// TwinCAT 3 PLC project RBB
// ProgramVersion: 3.1.4024.0
// libraries:
//   Tc2_Standard, * (Beckhoff Automation GmbH)
//   Tc2_System, * (Beckhoff Automation GmbH)
//   Tc3_Module, * (Beckhoff Automation GmbH)
// project tree:
//   DUTs/ E_ClientServerSteps.TcDUT, GPSReceive.TcDUT, ST_FrameFifoEntry.TcDUT, ST_FrameFifoEntrydata.TcDUT, ST_FrameFifoEntrydatarx.TcDUT, ST_FrameFifoEntrydata_1.TcDUT, ST_FrameFifoEntrydata_2.TcDUT, Union_LREAL.TcDUT, Union_LREAL_STRING.TcDUT, Union_REAL.TcDUT, Union_STRING_10.TcDUT, Union_STRING_2.TcDUT, Union_STRING_3.TcDUT, Union_STRING_4.TcDUT, Union_UDINT.TcDUT, Union_UINT.TcDUT, Union_WORD.TcDUT
//   GVLs/ GVL.TcGVL
//   / PlcTask.TcTTO
//   POUs/Background/ Background.TcPOU
//   POUs/Communication/ FB_AHRSCommunication.TcPOU, FB_ESCcommunication.TcPOU, FB_GPSCommunication.TcPOU
//   POUs/FUCTION BLOCK/UDP Source/ FB_FrameFifo.TcPOU, FB_FrameFiforx.TcPOU, FB_FrameFifo_1.TcPOU, FB_FrameFifo_2.TcPOU, FB_LogFifo.TcPOU, FB_PeerToPeer.TcPOU, FB_PeerToPeer_1.TcPOU, FB_PeerToPeer_2.TcPOU
//   POUs/FUNCTION/ FC_AnalogRead.TcPOU, FC_BatCalculate.TcPOU, FC_CalculateAzimuth.TcPOU, FC_HaversineDistance.TcPOU, FC_HMIRead.TcPOU
//   POUs/ MAIN.TcPOU, UDPCommunication_RBB.TcPOU
//   POUs/Module/ ESC.TcPOU, RelayModule.TcPOU
//   POUs/Sensor/ AHRS.TcPOU, GPS.TcPOU, LeakSensor.TcPOU
// real-time tasks:
//   TASK PlcTask: cycle T#10ms, priority 20, ADS port 350

CONFIGURATION RBB
    RESOURCE PLC ON TwinCAT3
        TASK PlcTask(INTERVAL := T#10ms, PRIORITY := 20);
        PROGRAM MAIN WITH PlcTask : MAIN;
    END_RESOURCE
END_CONFIGURATION

// ---- DUTs/E_ClientServerSteps.TcDUT
TYPE E_ClientServerSteps :
(
	eUDP_STATE_IDLE		:= 0,
	eUDP_STATE_CREATE_START,
	eUDP_STATE_CREATE_WAIT,
	eUDP_STATE_SEND_START,
	eUDP_STATE_SEND_WAIT,
	eUDP_STATE_RECEIVE_START,
	eUDP_STATE_RECEIVE_WAIT,
	eUDP_STATE_CLOSE_START,
	eUDP_STATE_CLOSE_WAIT,
	eUDP_STATE_ERROR
);
END_TYPE

// ---- DUTs/GPSReceive.TcDUT
TYPE GPSReceive :
UNION
	value : STRING;
	packed : ARRAY[0..69] OF BYTE;
END_UNION
END_TYPE

// ---- DUTs/ST_FrameFifoEntry.TcDUT
TYPE ST_FrameFifoEntry :
STRUCT
	 caseSelector : INT;              // Selector to choose the active structure
    data         : U_FrameFifoEntrydata;
END_STRUCT
END_TYPE

// ---- DUTs/ST_FrameFifoEntrydata.TcDUT
TYPE ST_FrameFifoEntrydata :
STRUCT
	stRemoteAddr 	: ST_SockAddr;
	txdata : ARRAY[0..TXDATASIZE] OF BYTE;	
END_STRUCT
END_TYPE

// ---- DUTs/ST_FrameFifoEntrydatarx.TcDUT
TYPE ST_FrameFifoEntrydatarx :
STRUCT
	stRemoteAddr 	: ST_SockAddr;
	rxdata : ARRAY[0..RXDATASIZE] OF BYTE;
END_STRUCT
END_TYPE

// ---- DUTs/ST_FrameFifoEntrydata_1.TcDUT
TYPE ST_FrameFifoEntrydata_1 :
STRUCT	
	stRemoteAddr 	: ST_SockAddr;
	txdata : ARRAY[0..TXDATASIZE_1] OF BYTE; 
END_STRUCT
END_TYPE

// ---- DUTs/ST_FrameFifoEntrydata_2.TcDUT
TYPE ST_FrameFifoEntrydata_2 :
STRUCT
	stRemoteAddr 	: ST_SockAddr;
	txdata : ARRAY[0..TXDATASIZE_2] OF BYTE; 
END_STRUCT
END_TYPE

// ---- DUTs/Union_LREAL.TcDUT
TYPE Union_LREAL :
UNION
	value : LREAL;
	packed : ARRAY[0..7] OF BYTE;
END_UNION
END_TYPE

// ---- DUTs/Union_LREAL_STRING.TcDUT
TYPE Union_LREAL_STRING :
UNION
	value : STRING;
	packed : ARRAY[0..7] OF BYTE;
END_UNION
END_TYPE

// ---- DUTs/Union_REAL.TcDUT
TYPE Union_REAL :
UNION
	value : REAL;
	Packed : ARRAY[0..3] OF BYTE;
END_UNION
END_TYPE

// ---- DUTs/Union_STRING_10.TcDUT
TYPE Union_STRING_10 :
UNION
	value : STRING;
	Packed : ARRAY[0..9] OF BYTE;
END_UNION
END_TYPE

// ---- DUTs/Union_STRING_2.TcDUT
TYPE Union_STRING_2 :
UNION
	value : STRING;
	Packed : ARRAY[0..1] OF BYTE;
END_UNION
END_TYPE

// ---- DUTs/Union_STRING_3.TcDUT
TYPE Union_STRING_3 :
UNION
	value : STRING;
	Packed : ARRAY[0..2] OF BYTE;
END_UNION
END_TYPE

// ---- DUTs/Union_STRING_4.TcDUT
TYPE Union_STRING_4 :
UNION
	value : STRING;
	Packed : ARRAY[0..3] OF BYTE;
END_UNION
END_TYPE

// ---- DUTs/Union_UDINT.TcDUT
TYPE Union_UDINT :
UNION
	value : UDINT ;
	packed : ARRAY[0..3] OF BYTE;
END_UNION
END_TYPE

// ---- DUTs/Union_UINT.TcDUT
TYPE Union_UINT :
UNION
	value : UINT;
	packed : ARRAY[0..1] OF BYTE;
END_UNION
END_TYPE

// ---- DUTs/Union_WORD.TcDUT
TYPE Union_WORD :
UNION
	value : WORD;
	packed : ARRAY[0..1] OF BYTE;
END_UNION
END_TYPE

// ---- GVLs/GVL.TcGVL
VAR_GLOBAL
	
	RxBufferEL6001		: ComBuffer;	
	TxBufferEL6001		: ComBuffer;	
	
	RxBufferEL6002	    : ComBuffer;	
	TxBufferEL6002		: ComBuffer;	
	
	RxBufferEL6021		: ComBuffer;	
	TxBufferEL6021		: ComBuffer;
	
	
	AI_00 AT%I* : WORD;
    AI_01 AT%I* : WORD;
	
	//Algorithm_Sw : BOOL;
 
 
	 
END_VAR

VAR_GLOBAL CONSTANT
 TXDATASIZE : INT := 101; // 59(60) , 23(24) , 17(18) , 101(102) , test 105(106)
 
 TXDATASIZE_1 : INT := 12; 
 TXDATASIZE_2 : INT := 15; 
 
 
 RXDATASIZE : INT := 1000; 
 
 
 PLCPRJ_BUFFER_SIZE					: UDINT := 1000;(* Max. internal fifo/receiver buffer size *)

(* Some project specific error codes *)
PLCPRJ_ERROR_SENDFIFO_OVERFLOW		: UDINT := 16#8103;
PLCPRJ_ERROR_RECFIFO_OVERFLOW		: UDINT := 16#8104;

END_VAR

// ---- POUs/MAIN.TcPOU
PROGRAM MAIN
VAR

// BAT

rBatvoltage : REAL; // UDP DATA
rBatcurrent : REAL; // UDP DATA
rBatWattsec : LREAL; 
AccumulatedBatData : LREAL :=0.0; // UDP DATA
lbatstate : LREAL; // UDP DATA

battimer : TON;

HMIbatV : STRING; // HMI
HMIbatA : STRING; // HMI
HMIbatW : STRING; // HMI
HMIbatS : STRING; // HMI

//AHRS

bAHRSError : BOOL;
AHRSErrorID : ComError_t;

HMIYAW : STRING;
HMIPITCH : STRING;
HMIROLL : STRING;

// ESC

bESCerror : BOOL;
ESCerrorID : ComError_t;
thrusterrightrpm : UINT;
thrusterleftrpm : UINT;


// GPS

bGPSrror : BOOL;
GPSErrorID : ComError_t;

GPSlat1 : LREAL;
GPSlon1 : LREAL;

HMILatitude : STRING;
HMILongitude : STRING;
HMISpeed : STRING;
	
// LEAK SENSOR

SystemLeakState : BOOL;
Leaksensorerror : BOOL;
Leaksensorerrorid : MODBUS_ERRORS;

// RELAY	
  
RelayModuledata : BYTE ;
RelayModuleError : BOOL;
RelayModuleErrorID : UDINT;

// UDP

UDPAlgorithm : INT;
UDPtimer : TON;


// Algorithm

    state : UINT := 0;
    timer : TON;
    stayTimer : TON;
    distance : LREAL;
    azimuth : LREAL;
   
    lat1, lon1, lat2, lon2, lat3, lon3, lat4, lon4 : LREAL;
	lat5, lon5, lat6, lon6, lat7, lon7, lat8, lon8,
	lat9, lon9, lat10, lon10, lat11, lon11, lat12, lon12,
	lat13, lon13, lat14, lon14, lat15, lon15, lat16, lon16 : LREAL;
	
    baseLat, baseLon : LREAL;
    currentTargetLat, currentTargetLon : LREAL;
    waypointIndex : UINT :=1;
	turnAngle : LREAL;
	turnangelzero : BOOL;
	esccontroltimer : TON;
	esccontroltimer1 : TON;
	esccontroltimer2 : TON;
	esccontroltimer3 : TON;
	esccontroltimer4 : TON;
		
	bturnangle : BOOL := TRUE;
	bturnangle2 : BOOL := TRUE;
	bstraight : BOOL := TRUE;
	bstop : BOOL := TRUE;
	
// Utilities

	bPCShutdown: BOOL;
	fbShutdown: NT_Shutdown;
	bShutdown: BOOL :=FALSE;
	
	step : INT;
	start : BOOL;
	Shutdown : BOOL := FALSE;
	
	i: INT;
END_VAR

// BAT 

rBatvoltage := FC_AnalogRead(selectData := AI_00, SelectRange := 600);
rBatcurrent := FC_AnalogRead(selectData := AI_01, SelectRange := 100);
rBatWattsec := (rBatvoltage*rBatcurrent)/3600;

IF NOT battimer.Q THEN
battimer(IN:=TRUE, PT := T#1S);
ELSE 
battimer(IN:=FALSE);
AccumulatedBatData := AccumulatedBatData + rBatWattsec;
END_IF

lbatstate := FC_BatCalculate(lbatdata := AccumulatedBatData);

HMIbatV := FC_HMIRead(linput := rBatvoltage, inumber := 2);
HMIbatA := FC_HMIRead(linput := rBatcurrent, inumber := 2);
HMIbatW := FC_HMIRead(linput := AccumulatedBatData , inumber := 2);
HMIbatS := FC_HMIRead(linput := lbatstate, inumber := 2);
 
// AHRS 

AHRS();
bAHRSError := AHRS.bAHRSError;
AHRSErrorID := AHRS.AHRSErrorID;

HMIYAW :=FC_HMIRead(linput := AHRS.ResultYAW, inumber := 1);
HMIPITCH :=FC_HMIRead(linput := AHRS.ResultPITCH, inumber := 1);
HMIROLL :=FC_HMIRead(linput := AHRS.ResultROLL, inumber := 1);

// ESC

ESC();
bESCerror := ESC.bESCerror;
ESCerrorID := ESC.ESCerrorID;

IF ESC.sMotorspeed = 'ESC1:1650' THEN
	thrusterrightrpm := 750;
ELSIF ESC.sMotorspeed = 'ESC1:1750' THEN
	thrusterrightrpm := 1250;
ELSIF  ESC.sMotorspeed = 'ESC1:1700' THEN
	thrusterrightrpm := 1000;
ELSIF ESC.sMotorspeed = 'ESC2:1350' THEN
	thrusterleftrpm := 750;
ELSIF  ESC.sMotorspeed = 'ESC2:1250' THEN
	thrusterleftrpm := 1250;
ELSIF  ESC.sMotorspeed = 'ESC2:1300' THEN
	thrusterleftrpm := 1000;
END_IF 


// GPS 

GPS();
bGPSrror := GPS.bGPSrror;
GPSErrorID := GPS.GPSErrorID;

GPSlat1 := GPS.gpslat;
GPSlon1 := GPS.gpslon;

HMILatitude :=FC_HMIRead(linput := GPS.gpslat, inumber := 1);
HMILongitude :=FC_HMIRead(linput := GPS.gpslon, inumber := 1);
HMISpeed :=FC_HMIRead(linput := GPS.gpsSpeedms, inumber := 1);

// LEAK SENSOR

LeakSensor();
SystemLeakState := LeakSensor.LeakSensorState;
Leaksensorerror := LeakSensor.Leaksensorerror;
Leaksensorerrorid := LeakSensor.leaksensorerrorid;
 
// RELAY Module

RelayModule();
RelayModuleError := RelayModule.RelayModuleError;
RelayModuleErrorID := RelayModule.RelayModuleErrorID;
RelayModuledata := RelayModule.relaymodulesendOnData;

// UDPCommunication

UDPCommunication_RBB();
	CASE UDPAlgorithm OF
		0 :
		IF UDPCommunication_RBB.UDPstart THEN
			IF UDPCommunication_RBB.Receiveaddress = 16#01 THEN
				UDPAlgorithm := 10;
			ELSIF UDPCommunication_RBB.Receiveaddress = 16#02 THEN
				UDPAlgorithm := 10;
			ELSIF UDPCommunication_RBB.Receiveaddress = 16#03 THEN
				UDPAlgorithm := 10;
			ELSIF UDPCommunication_RBB.Receiveaddress = 16#04 THEN
				UDPAlgorithm := 10;
			END_IF		
		END_IF
		
		10 :
		 UDPCommunication_RBB.UDPstart := FALSE;
		 UDPtimer(IN:= TRUE, PT:= T#1S);
		 IF UDPtimer.Q THEN
		 UDPCommunication_RBB.UDPstart3 := TRUE;
		 UDPtimer(IN:= FALSE);
		 UDPAlgorithm := 20;
		 END_IF
		 		 		 
		 20 :
		 UDPtimer(IN:= TRUE, PT:= T#1S);
		 IF UDPtimer.Q THEN
		 UDPCommunication_RBB.UDPstart3 := FALSE;	
         UDPtimer(IN:= FALSE);
		 UDPAlgorithm := 30; 
		 END_IF
		 		 
		 30 : 
		 UDPtimer(IN:= TRUE, PT:= T#1S);
		 IF UDPtimer.Q THEN
		  IF UDPCommunication_RBB.Receiveaddress = 16#03 THEN
			UDPCommunication_RBB.UDPstart2 := TRUE;
			UDPtimer(IN:= FALSE);
		    UDPAlgorithm := 40;
		  ELSE
		  UDPCommunication_RBB.UDPstart := TRUE;		
		  UDPCommunication_RBB.bSendOnceToRemote2 := FALSE;
		  UDPtimer(IN:= FALSE);
		  UDPAlgorithm := 0;
		  END_IF
		 END_IF
		 
		 40 :
		 UDPtimer(IN:= TRUE, PT:= T#1S);
		 IF UDPtimer.Q THEN
		 UDPCommunication_RBB.UDPstart2 := FALSE;	
         UDPtimer(IN:= FALSE);
		 UDPAlgorithm := 50; 
		 END_IF
		 
		 50 :
		 UDPtimer(IN:= TRUE, PT:= T#1S);
		 IF UDPtimer.Q THEN
		 UDPCommunication_RBB.UDPstart := TRUE;
		 UDPCommunication_RBB.bSendOnceToRemote1 := FALSE;
		 UDPtimer(IN:= FALSE);
		 UDPAlgorithm := 0;
		 END_IF
	END_CASE


// Algorithm

IF UDPCommunication_RBB.Algorithmstop THEN	

  IF UDPCommunication_RBB.Algorithm_Sw THEN
    CASE state OF
        0: // Start algorithm, initialize first target
		    lat1 := UDPCommunication_RBB.packetwetpointlat1.value;
			lon1 := UDPCommunication_RBB.packetwetpointlot1.value;
            currentTargetLat := lat1;
            currentTargetLon := lon1;
            state := 10;
			

        10: // Calculate distance to the current target
            distance := FC_HaversineDistance(GPS.gpslat, GPS.gpslon, currentTargetLat, currentTargetLon);
            IF ABS(distance) <=10 THEN
                state := 13; // Go to the stay state if already within 10m
            ELSE
                timer(IN := TRUE, PT := T#1S);
                IF timer.Q THEN
                    state := 11;
                    timer(IN := FALSE); // Reset timer
                END_IF
            END_IF

        11: // Calculate azimuth and move
            azimuth := FC_CalculateAzimuth(GPS.gpslat, GPS.gpslon, currentTargetLat, currentTargetLon);
            turnAngle := azimuth - UDPCommunication_RBB.packetahrsheading.value;
			
            IF turnAngle > 180 THEN
                turnAngle := turnAngle - 360;
            ELSIF turnAngle < -180 THEN
                turnAngle := turnAngle + 360;
            END_IF
			
			IF ABS(turnAngle) <= 25 THEN  
                 state := 12; 
											
            ELSIF turnAngle > 0 THEN// Turn right
			   IF bturnangle THEN
				ESC.sMotorspeed := 'ESC2:1250'; //62.5%
				esccontroltimer2(IN:=TRUE, PT:=T#1S);
				 IF esccontroltimer2.Q THEN
				   ESC.sMotorspeed := 'ESC1:1650';	// 37.5%			   
				   esccontroltimer2(IN:=FALSE);
                   bturnangle := FALSE;				   
				 END_IF 			
				END_IF 
											
            ELSE// Turn left	
				 IF bturnangle2 THEN
				  ESC.sMotorspeed := 'ESC1:1750'; //62.5% 
				 esccontroltimer4(IN:=TRUE, PT:=T#1S);
				  IF esccontroltimer4.Q THEN
				   ESC.sMotorspeed := 'ESC2:1350'; //37.5%
				   esccontroltimer4(IN:=FALSE);
                   bturnangle2 := FALSE;				   
				  END_IF 			
				END_IF 
		  END_IF 
             				        
			
									
		12 : // Move
		
		distance := FC_HaversineDistance(GPS.gpslat, GPS.gpslon, currentTargetLat, currentTargetLon);
		azimuth := FC_CalculateAzimuth(GPS.gpslat, GPS.gpslon, currentTargetLat, currentTargetLon);
        turnAngle := azimuth - UDPCommunication_RBB.packetahrsheading.value;
			
            IF turnAngle > 180 THEN
                turnAngle := turnAngle - 360;
            ELSIF turnAngle < -180 THEN
                turnAngle := turnAngle + 360;
            END_IF
			
			
		
            IF ABS(turnAngle) <= 25 THEN  
			IF bstraight THEN
				ESC.sMotorspeed := 'ESC2:1300'; //50%
				esccontroltimer1(IN:=TRUE, PT:=T#1S);
				 IF esccontroltimer1.Q THEN
				   ESC.sMotorspeed := 'ESC1:1700'; // 50%
				   esccontroltimer1(IN:=FALSE);
                   bstraight := FALSE;				   
				 END_IF 	
                  ELSIF ABS(distance) <=10 THEN		         
				   esccontroltimer3(IN:=TRUE, PT:=T#1S);
				   IF esccontroltimer3.Q THEN	   
				   ESC.sMotorspeed := 'stop';			   
				   esccontroltimer3(IN:=FALSE);				
				   state := 13;	
				   END_IF
			  END_IF  
              ELSE
                   state :=11;	
	               bstraight := TRUE;
				   bturnangle := TRUE;	
				   bturnangle2 := TRUE;	
              END_IF	


        13: // Check distance again
            stayTimer(IN := TRUE, PT := T#30S);
            IF stayTimer.Q THEN
				ESC.sMotorspeed := '';
				   bstraight := TRUE;
				   bturnangle := TRUE;	
				   bturnangle2 := TRUE;	
                state := 14; // Next waypoint or finish
                stayTimer(IN := FALSE); // Reset stay timer
            END_IF
           


        14: // Check if there are more waypoints to visit
		    //waypointIndex 
            CASE waypointIndex OF
                1:
				    lat2 := UDPCommunication_RBB.packetwetpointlat2.value;
					lon2 := UDPCommunication_RBB.packetwetpointlot2.value;
                    currentTargetLat := lat2;
                    currentTargetLon := lon2;
                    waypointIndex := 2;
                    state := 10;
                2:
				    lat3 := UDPCommunication_RBB.packetwetpointlat3.value;
					lon3 := UDPCommunication_RBB.packetwetpointlot3.value;
                    currentTargetLat := lat3;
                    currentTargetLon := lon3;
                    waypointIndex := 3;
                    state := 10;
                3:
				    lat4 := UDPCommunication_RBB.packetwetpointlat4.value;
					lon4 := UDPCommunication_RBB.packetwetpointlot4.value;
                    currentTargetLat := lat4;
                    currentTargetLon := lon4;
                    waypointIndex := 4;
                    state := 10;
                4:
				    lat5 := UDPCommunication_RBB.packetwetpointlat4.value;
					lon5 := UDPCommunication_RBB.packetwetpointlot4.value;
                    currentTargetLat := lat5;
                    currentTargetLon := lon5;
                    waypointIndex := 5;
                    state := 10;
				5:
				    lat6 := UDPCommunication_RBB.packetwetpointlat4.value;
					lon6 := UDPCommunication_RBB.packetwetpointlot4.value;
                    currentTargetLat := lat6;
                    currentTargetLon := lon6;
                    waypointIndex := 6;
                    state := 10;
				6:
				    lat7 := UDPCommunication_RBB.packetwetpointlat4.value;
					lon7 := UDPCommunication_RBB.packetwetpointlot4.value;
                    currentTargetLat := lat7;
                    currentTargetLon := lon7;
                    waypointIndex := 7;
                    state := 10;
				7:
				    lat8 := UDPCommunication_RBB.packetwetpointlat4.value;
					lon8 := UDPCommunication_RBB.packetwetpointlot4.value;
                    currentTargetLat := lat8;
                    currentTargetLon := lon8;
                    waypointIndex := 8;
                    state := 10;
				8:
				    lat9 := UDPCommunication_RBB.packetwetpointlat4.value;
					lon9 := UDPCommunication_RBB.packetwetpointlot4.value;
                    currentTargetLat := lat9;
                    currentTargetLon := lon9;
                    waypointIndex := 9;
                    state := 10;
				9:
				    lat10 := UDPCommunication_RBB.packetwetpointlat4.value;
					lon10 := UDPCommunication_RBB.packetwetpointlot4.value;
                    currentTargetLat := lat10;
                    currentTargetLon := lon10;
                    waypointIndex := 10;
                    state := 10;
				10:
				    lat11 := UDPCommunication_RBB.packetwetpointlat4.value;
					lon11 := UDPCommunication_RBB.packetwetpointlot4.value;
                    currentTargetLat := lat11;
                    currentTargetLon := lon11;
                    waypointIndex := 11;
                    state := 10;
				11:
				    lat12 := UDPCommunication_RBB.packetwetpointlat4.value;
					lon12 := UDPCommunication_RBB.packetwetpointlot4.value;
                    currentTargetLat := lat12;
                    currentTargetLon := lon12;
                    waypointIndex := 12;
                    state := 10;
				12:
				    lat13 := UDPCommunication_RBB.packetwetpointlat4.value;
					lon13 := UDPCommunication_RBB.packetwetpointlot4.value;
                    currentTargetLat := lat13;
                    currentTargetLon := lon13;
                    waypointIndex := 13;
                    state := 10;
				13:
				    lat14 := UDPCommunication_RBB.packetwetpointlat4.value;
					lon14 := UDPCommunication_RBB.packetwetpointlot4.value;
                    currentTargetLat := lat14;
                    currentTargetLon := lon14;
                    waypointIndex := 14;
                    state := 10;
				14:
				    lat15 := UDPCommunication_RBB.packetwetpointlat4.value;
					lon15 := UDPCommunication_RBB.packetwetpointlot4.value;
                    currentTargetLat := lat15;
                    currentTargetLon := lon15;
                    waypointIndex := 15;
                    state := 10;
				15:
				    lat16 := UDPCommunication_RBB.packetwetpointlat4.value;
					lon16 := UDPCommunication_RBB.packetwetpointlot4.value;
                    currentTargetLat := lat16;
                    currentTargetLon := lon16;
                    waypointIndex := 16;
                    state := 10;  
 
                 16 :  
                    state := 20;
            END_CASE	 
                 20: 
		        ESC.sMotorspeed := 'stop';
				 
	 			
    END_CASE
ELSE
    // Reset state and timers if Algorithm_sw is turned off
    state := 0;
    timer(IN := FALSE);
    stayTimer(IN := FALSE);
    waypointIndex := 1; // Reset waypoint index
END_IF 

ELSE
	esc.sMotorspeed := 'stop';
END_IF


// Utilities
shutdown := UDPCommunication_RBB.controlshutdown;
IF Shutdown THEN
	bShutdown := TRUE;
END_IF
fbShutdown(
NETID:= , 
DELAY:= 5, 
START:= bShutdown, 
TMOUT:= , 
BUSY=> , 
ERR=> , 
ERRID=> );

END_PROGRAM

// ---- POUs/FUNCTION/FC_AnalogRead.TcPOU
FUNCTION FC_AnalogRead : REAL
VAR_INPUT
	SelectData : WORD;
	SelectRange : INT;
END_VAR
VAR
	Transdata : REAL;
END_VAR

Transdata := WORD_TO_REAL(selectData);
// FC_AnalogRead :=(Transdata*SelectRange)/32767;
FC_AnalogRead :=(Transdata/32767)*SelectRange;

END_FUNCTION

// ---- POUs/FUNCTION/FC_BatCalculate.TcPOU
FUNCTION FC_BatCalculate : LREAL
VAR_INPUT
	lbatdata : LREAL;
END_VAR
VAR
END_VAR

FC_BatCalculate := ((3000-lbatdata)/3000)*100; // 1000 UDP

END_FUNCTION

// ---- POUs/FUNCTION/FC_HMIRead.TcPOU
FUNCTION FC_HMIRead : STRING
VAR_INPUT
	linput : LREAL;
	inumber : INT;
END_VAR
VAR
END_VAR

FC_HMIRead := LREAL_TO_FMTSTR(linput,inumber,TRUE);

END_FUNCTION

// ---- POUs/Sensor/AHRS.TcPOU
PROGRAM AHRS
VAR
	fbAHRSCommunication : FB_AHRSCommunication;
	ahrsdatayaw, ahrsdatapitch, ahrsdataroll : Union_REAL;
	ResultYAW, ResultPITCH, ResultROLL : REAL;
	bAHRSError : BOOL;
    AHRSErrorID : ComError_t;
END_VAR

fbAHRSCommunication(TxBuffer:=TxBufferEL6001, RxBuffer:=RxBufferEL6001,
bReceiveError => bAHRSError, eReceiveErrorID =>AHRSErrorID );

ahrsdatayaw.Packed[0] := Background.stIn_EL6001.D[4];
ahrsdatayaw.Packed[1] := Background.stIn_EL6001.D[5];
ahrsdatayaw.Packed[2] := Background.stIn_EL6001.D[6];
ahrsdatayaw.Packed[3] := Background.stIn_EL6001.D[7];
ResultYAW := ahrsdatayaw.value;


ahrsdatapitch.Packed[0] := Background.stIn_EL6001.D[8];
ahrsdatapitch.Packed[1] := Background.stIn_EL6001.D[9];
ahrsdatapitch.Packed[2] := Background.stIn_EL6001.D[10];
ahrsdatapitch.Packed[3] := Background.stIn_EL6001.D[11];
ResultPITCH := ahrsdatapitch.value;


ahrsdataroll.Packed[0] := Background.stIn_EL6001.D[12];
ahrsdataroll.Packed[1] := Background.stIn_EL6001.D[13];
ahrsdataroll.Packed[2] := Background.stIn_EL6001.D[14];
ahrsdataroll.Packed[3] := Background.stIn_EL6001.D[15];
ResultROLL := ahrsdatapitch.value;

END_PROGRAM

// ---- POUs/Communication/FB_AHRSCommunication.TcPOU
FUNCTION_BLOCK FB_AHRSCommunication
VAR_IN_OUT
	TxBuffer	: ComBuffer;
	RxBuffer	: ComBuffer;
END_VAR

VAR_INPUT
END_VAR
VAR_OUTPUT
	bReceiveError	: BOOL;
	eReceiveErrorID	: ComError_t;
END_VAR
VAR
	Timer		: TON := (PT:=T#1S);
	fbSend		: SendString;
	bSendBusy	: BOOL;
    eSendErrorID: ComError_t;
	fbReceive		: ReceiveString;
	sReceivedString	: STRING;
	sLastReceivedString: STRING;
	bStringReceived	: BOOL;
	bReceiveBusy	: BOOL;
	bReceiveTimeout	: BOOL;
	nReceiveCounter	: UDINT;
END_VAR

Timer(IN:=TRUE);
IF Timer.Q OR fbSend.Busy THEN
	Timer(IN:=FALSE); (* reset timer *)
	fbSend(	SendString:= '',
			TXbuffer:= TxBuffer,
			Busy=> bSendBusy,
			Error=> );
	IF fbSend.Error <> COMERROR_NOERROR THEN
		eSendErrorID := fbSend.Error;
	END_IF
END_IF

fbReceive(
	Prefix:='',
	Suffix:= '',
	Timeout:= T#1s,
	ReceivedString:= sReceivedString,
	RXbuffer:= RxBuffer,
	StringReceived=> bStringReceived,
	Busy=> bReceiveBusy,
	Error=> ,
	RxTimeout=> bReceiveTimeout );
	
  IF fbReceive.Error <> COMERROR_NOERROR THEN
	 eReceiveErrorID := fbReceive.Error;
  END_IF

  IF bStringReceived THEN
	nReceiveCounter := nReceiveCounter + 1;
	sLastReceivedString := sReceivedString;
  END_IF

END_FUNCTION_BLOCK

// ---- POUs/Background/Background.TcPOU
PROGRAM Background
VAR
	
	fbEL6001Ctrl		: SerialLineControl;
	bEL6001CtrlError	: BOOL;
	eEL6001CtrlErrorID	: ComError_t;
	
	fbEL6002Ctrl		: SerialLineControl;
	bEL6002CtrlError	: BOOL;
	eEL6002CtrlErrorID	: ComError_t;
	
	fbEL6021Ctrl		: SerialLineControl;
	bEL6021CtrlError	: BOOL;
	eEL6021CtrlErrorID	: ComError_t;
	
END_VAR

VAR_OUTPUT
	stIn_EL6001 AT %I*	: EL6inData22B;	
	stOut_EL6001 AT %Q*	: EL6outData22B;
	
	stIn_EL6002 AT %I*	: EL6inData22B;	
	stOut_EL6002 AT %Q*	: EL6outData22B;
	
	stIn_EL6021 AT %I*	: EL6inData22B;	
	stOut_EL6021 AT %Q*	: EL6outData22B;
END_VAR


fbEL6001Ctrl(
	Mode:= SERIALLINEMODE_EL6_22B, 
	pComIn:= ADR(stIn_EL6001), 
	pComOut:= ADR(stOut_EL6001), 
	SizeComIn:= SIZEOF(stIn_EL6001), 
	Error=> , 
	ErrorID=> , 
	TxBuffer:= TxBufferEL6001, 
	RxBuffer:= RxBufferEL6001 );
	
IF fbEL6001Ctrl.Error THEN
	bEL6001CtrlError := TRUE;
	eEL6001CtrlErrorID := fbEL6001Ctrl.ErrorID;
END_IF

fbEL6002Ctrl(
	Mode:= SERIALLINEMODE_EL6_22B, 
	pComIn:= ADR(stIn_EL6002), 
	pComOut:= ADR(stOut_EL6002), 
	SizeComIn:= SIZEOF(stIn_EL6002), 
	Error=> , 
	ErrorID=> , 
	TxBuffer:= TxBufferEL6002, 
	RxBuffer:= RxBufferEL6002 );
	
IF fbEL6002Ctrl.Error THEN
	bEL6002CtrlError := TRUE;
	eEL6002CtrlErrorID := fbEL6002Ctrl.ErrorID;
END_IF

fbEL6021Ctrl(
	Mode:= SERIALLINEMODE_EL6_22B, 
	pComIn:= ADR(stIn_EL6021), 
	pComOut:= ADR(stOut_EL6021), 
	SizeComIn:= SIZEOF(stIn_EL6021), 
	Error=> , 
	ErrorID=> , 
	TxBuffer:= TxBufferEL6021, 
	RxBuffer:= RxBufferEL6021 );
IF fbEL6021Ctrl.Error THEN
	bEL6021CtrlError := TRUE;
	eEL6021CtrlErrorID := fbEL6021Ctrl.ErrorID;
END_IF

END_PROGRAM

// ---- POUs/Module/ESC.TcPOU
PROGRAM ESC
VAR_INPUT
	
	sMotorspeed : STRING; // 'ESC1:value', 'ESC2:value'

END_VAR
VAR_OUTPUT
	
END_VAR
VAR
	fbescCommunication : FB_ESCcommunication;

	bESCerror : BOOL;
    ESCerrorID : ComError_t;
	
	currentcotrol : UINT :=0;
	previouscotrol : UINT :=0;
	timer: TON;
	
	
END_VAR

fbescCommunication(senddata := sMotorspeed, TxBuffer:=TxBufferEL6021, RxBuffer:=RxBufferEL6021,
bReceiveError => bESCerror, eReceiveErrorID =>ESCerrorID);

END_PROGRAM

// ---- POUs/Communication/FB_ESCcommunication.TcPOU
FUNCTION_BLOCK FB_ESCcommunication
VAR_INPUT
	
senddata : STRING;

END_VAR

VAR_IN_OUT
	TxBuffer	: ComBuffer;
	RxBuffer	: ComBuffer;
END_VAR
VAR_OUTPUT
	bReceiveError	: BOOL;
	eReceiveErrorID	: ComError_t;
END_VAR
VAR
	Timer		: TON := (PT:=T#1S);
	fbSend		: SendString;
	bSendBusy	: BOOL;
	eSendErrorID: ComError_t;

	fbReceive		: ReceiveString;
	sReceivedString	: STRING;
	sLastReceivedString: STRING;
	bStringReceived	: BOOL;
	bReceiveBusy	: BOOL;
	bReceiveTimeout	: BOOL;
	nReceiveCounter	: UDINT;
END_VAR

Timer(IN:=TRUE);
IF Timer.Q OR fbSend.Busy THEN
	Timer(IN:=FALSE); (* reset timer *)
	fbSend(	SendString:= senddata,
			TXbuffer:= TxBuffer,
			Busy=> bSendBusy,
			Error=> );
	IF fbSend.Error <> COMERROR_NOERROR THEN
		eSendErrorID := fbSend.Error;
	END_IF
END_IF

fbReceive(
	Prefix:= '',
	Suffix:= '',
	Timeout:= T#1s,
	ReceivedString:= sReceivedString,
	RXbuffer:= RxBuffer,
	StringReceived=> bStringReceived,
	Busy=> bReceiveBusy,
	Error=> ,
	RxTimeout=> bReceiveTimeout );
IF fbReceive.Error <> COMERROR_NOERROR THEN
	eReceiveErrorID := fbReceive.Error;
END_IF
IF bStringReceived THEN
	nReceiveCounter := nReceiveCounter + 1;
	sLastReceivedString := sReceivedString;
END_IF

END_FUNCTION_BLOCK

// ---- POUs/Sensor/GPS.TcPOU
PROGRAM GPS
VAR
	fbGPSCommunication : FB_GPSCommunication;
	GpsRXdata : GPSReceive;
	gpslat1 : Union_STRING_2;
	gpslat2 : Union_STRING_10;
	gpslon1 : Union_STRING_3;
	gpslon2 : Union_STRING_10;
	gpsSpeed1 : Union_STRING_3;
	gpslati,gpslatd,gpslat : LREAL;
	gpsloni,gpslond,gpslon : LREAL;
	gpsSpeedknots,gpsSpeedms : LREAL;
	bGPSrror : BOOL;
    GPSErrorID : ComError_t;
END_VAR

fbGPSCommunication(TxBuffer:=TxBufferEL6002, RxBuffer:=RxBufferEL6002,
bReceiveError => bGPSrror, eReceiveErrorID =>GPSErrorID);
GpsRXdata.value := fbGPSCommunication.sReceivedString ;

gpslat1.Packed[0] :=  GpsRXdata.packed[19];
gpslat1.Packed[1] :=  GpsRXdata.packed[20];
gpslati := STRING_TO_LREAL(gpslat1.value);

gpslat2.Packed[0] := GpsRXdata.packed[21];
gpslat2.Packed[1] := GpsRXdata.packed[22];
gpslat2.Packed[2] := GpsRXdata.packed[23];
gpslat2.Packed[3] := GpsRXdata.packed[24];
gpslat2.Packed[4] := GpsRXdata.packed[25];
gpslat2.Packed[5] := GpsRXdata.packed[26];
gpslat2.Packed[6] := GpsRXdata.packed[27];
gpslat2.Packed[7] := GpsRXdata.packed[28];
gpslat2.Packed[8] := GpsRXdata.packed[29];
gpslat2.Packed[9] := GpsRXdata.packed[30];

gpslatd := STRING_TO_LREAL(gpslat2.value)/60;

gpslat := gpslati + gpslatd ;

gpslon1.Packed[0] := GpsRXdata.packed[34];
gpslon1.Packed[1] := GpsRXdata.packed[35];
gpslon1.Packed[2] := GpsRXdata.packed[36];
gpsloni := STRING_TO_LREAL(gpslon1.value);


gpslon2.Packed[0] := GpsRXdata.packed[37];
gpslon2.Packed[1] := GpsRXdata.packed[38];
gpslon2.Packed[2] := GpsRXdata.packed[39];
gpslon2.Packed[3] := GpsRXdata.packed[40];
gpslon2.Packed[4] := GpsRXdata.packed[41];
gpslon2.Packed[5] := GpsRXdata.packed[42];
gpslon2.Packed[6] := GpsRXdata.packed[43];
gpslon2.Packed[7] := GpsRXdata.packed[44];
gpslon2.Packed[8] := GpsRXdata.packed[45];
gpslon2.Packed[9] := GpsRXdata.packed[46];

gpslond :=STRING_TO_LREAL(gpslon2.value)/60;

gpslon := gpsloni + gpslond;

gpsspeed1.Packed[0] := GpsRXdata.packed[50];
gpsspeed1.Packed[1] := GpsRXdata.packed[51];
gpsspeed1.Packed[2] := GpsRXdata.packed[52];

gpsspeedknots := STRING_TO_LREAL(gpsspeed1.value);
gpsspeedms := gpsspeedknots * 1.943;

END_PROGRAM

// ---- POUs/Communication/FB_GPSCommunication.TcPOU
FUNCTION_BLOCK FB_GPSCommunication
VAR_IN_OUT
	TxBuffer	: ComBuffer;
	RxBuffer	: ComBuffer;
END_VAR

VAR_OUTPUT
	sReceivedString	: STRING;
	bReceiveError	: BOOL;
	eReceiveErrorID	: ComError_t;
END_VAR

VAR
	Timer		: TON := (PT:=T#1S);
	fbSend		: SendString;
	bSendBusy	: BOOL;
	eSendErrorID: ComError_t;
	fbReceive		: ReceiveString;
	sLastReceivedString: STRING;
	bStringReceived	: BOOL;
	bReceiveBusy	: BOOL;

	bReceiveTimeout	: BOOL;
	nReceiveCounter	: UDINT;
END_VAR


Timer(IN:=TRUE);
IF Timer.Q OR fbSend.Busy THEN
	Timer(IN:=FALSE); (* reset timer *)
	fbSend(	SendString:= ,
			TXbuffer:= TxBuffer,
			Busy=> bSendBusy,
			Error=> );
	IF fbSend.Error <> COMERROR_NOERROR THEN
		eSendErrorID := fbSend.Error;
	END_IF
END_IF


fbReceive(
	Prefix:='$24',
	Suffix:= '$2a',
	Timeout:= T#1s,
	ReceivedString:= sReceivedString,
	RXbuffer:= RxBuffer,
	StringReceived=> bStringReceived,
	Busy=> bReceiveBusy,
	Error=> ,
	RxTimeout=> bReceiveTimeout );
IF fbReceive.Error <> COMERROR_NOERROR THEN
	eReceiveErrorID := fbReceive.Error;
END_IF
IF bStringReceived THEN
	nReceiveCounter := nReceiveCounter + 1;
	sLastReceivedString := sReceivedString;
END_IF

END_FUNCTION_BLOCK

// ---- POUs/Sensor/LeakSensor.TcPOU
PROGRAM LeakSensor
VAR
	leaksensorread: ModbusRtuMasterV2_KL6x22B;
	leakreceivedata : INT ;
	leakclock : TON;
    leaksensorerrorid : MODBUS_ERRORS;
	Leaksensorerror : BOOL;   
    leakstatetimer : TON; 
    LeakSensordata : BYTE; // UDP DATA
END_VAR

VAR_OUTPUT
	 
	 LeakSensorState : BOOL;
END_VAR

IF NOT leakclock.Q THEN
 leakclock(IN:=	TRUE, PT := T#1S);
 ELSE 
	 leakclock(IN:=FALSE);
 END_IF

	leaksensorread.ReadInputRegs(
	UnitID:= 1 , 
	Quantity:= 1, 
	MBAddr:= 16#0000 , 
	cbLength:= SIZEOF(leakreceivedata), 
	pMemoryAddr:= ADR(leakreceivedata), 
	AuxQuantity:= , 
	AuxMBAddr:= , 
	AuxcbLength:= , 
	pAuxMemoryAddr:= , 
	Execute:= leakclock.Q  , 
	Timeout:= T#1S, 
	BUSY=> , 
	Error=> Leaksensorerror, 
	ErrorId=>leaksensorerrorid , 
	cbRead=> ); 
	
LeakSensordata := LeakSensor.leaksensorread.InData.D[4] ;
  IF LeakSensordata =0 THEN    
     LeakSensorState := FALSE;
   ELSE
     LeakSensorState := TRUE;
   END_IF;

END_PROGRAM

// ---- POUs/Module/RelayModule.TcPOU
PROGRAM RelayModule
VAR
	relaysendcoil: FB_MBWriteCoils;
	relaysendOnData :  BYTE; //:= 16#04;  // 16#04 ON 3CH
	relayclock : TON;
	RelayModuleError : BOOL;
    RelayModuleErrorID : UDINT;
	
	CH1on : BOOL ; // HMI
CH1off : BOOL ; // HMI
CH1state : BOOL := FALSE; // HMI
	
CH2on : BOOL ; // HMI
CH2off : BOOL ; // HMI
CH2state : BOOL := FALSE; // HMI
	
CH3on : BOOL ; // HMI
CH3off : BOOL ; // HMI
CH3state : BOOL := FALSE; // HMI
	
CH4on : BOOL ; // HMI
CH4off : BOOL ; // HMI
CH4state : BOOL := FALSE; // HMI
	
CH5on : BOOL ; // HMI
CH5off : BOOL ; // HMI
CH5state : BOOL := FALSE; // HMI

	relaymodulesendOnData: BYTE;//:= 16#04;  // 16#04 ON 3CH
END_VAR

IF NOT relayclock.Q THEN
	relayclock(IN:=TRUE, PT := T#4S);
	ELSE 
		relayclock(IN:=FALSE);
	END_IF 


relaysendcoil(
	sIPAddr:= '192.168.10.134', 
	nTCPPort:= 502 , 
	nUnitID:= 1, 
	nQuantity:= 6 , 
	nMBAddr:= 16#0011 , 
	cbLength:=SIZEOF(relaymodulesendOnData) , 
	pSrcAddr:= ADR(relaymodulesendOnData), 
	bExecute:= relayclock.Q, 
	tTimeout:= T#2S, 
	bBusy=> , 
	bError=> RelayModuleError, 
	nErrId=> RelayModuleErrorID); 
	
	
	IF CH1on THEN
		relaymodulesendOnData := relaymodulesendOnData+16#01;
		CH1on := FALSE;
		CH1State := TRUE;
		END_IF
	IF CH1off THEN
	   relaymodulesendOnData := relaymodulesendOnData-16#01;
	   CH1off := FALSE;
	   CH1state := FALSE;
		END_IF
	
	IF CH2on THEN
		relaymodulesendOnData := relaymodulesendOnData+16#02;
		CH2on := FALSE;
		CH2State := TRUE;
		END_IF
	IF CH2off THEN
	    relaymodulesendOnData := relaymodulesendOnData-16#02;
		CH2off := FALSE;
		CH2state := FALSE;
		END_IF
		
	IF CH3on THEN
		relaymodulesendOnData := relaymodulesendOnData+16#04;
		CH3on := FALSE;
		CH3State := TRUE;
		END_IF
	IF CH3off THEN
	    relaymodulesendOnData := relaymodulesendOnData-16#04;
		CH3off := FALSE;
		CH3state := FALSE;
		END_IF
		
	IF CH4on THEN
		relaymodulesendOnData := relaymodulesendOnData+16#08;
		CH4on := FALSE;
		CH4State := TRUE;
		END_IF
	IF CH4off THEN
	    relaymodulesendOnData := relaymodulesendOnData-16#08;
		CH4off := FALSE;
		CH4state := FALSE;
		END_IF
		
	IF CH5on THEN
		relaymodulesendOnData := relaymodulesendOnData+16#10;
		CH5on := FALSE;
		CH5State := TRUE;
		END_IF
	IF CH5off THEN
	    relaymodulesendOnData := relaymodulesendOnData-16#10;
		CH5off := FALSE;
		CH5state := FALSE;
		END_IF

END_PROGRAM

// ---- POUs/UDPCommunication_RBB.TcPOU
PROGRAM UDPCommunication_RBB
VAR	
	bSendOnceToRemote	: BOOL := FALSE;(* Rising edge at this variable sends message to the remote host/port *)
	
	sSrvNetId			: T_AmsNetID 	:= '';(* TwinCAT TCP/IP server network address. Default: empty string. *)
	sLocalHost			: T_IPv4Addr 	:= '192.168.10.30';(* Local address: String containing an (Ipv4) Internet Protocol dotted address. *) 
	nLocalPort			: UDINT			:= 53635;(* Local address: IP port number *)//225
	sRemoteHost			: T_IPv4Addr 	:= '192.168.1.10'; //'192.168.1.10';(* Remote address: String containing an (Ipv4) Internet Protocol dotted address. *)
	nRemotePort			: UDINT 		:= 53634;(* Remote address: IP port number. *)//225
	bEnable				: BOOL 			:= TRUE;(* TRUE => Enable/connect, FALSE => Disable/disconnect *)
	bLog				: BOOL			:= TRUE;(* TRUE => Enable log message output, FALSE => Disable *)
	
	fbPeerToPeer		: FB_PeerToPeer := ( sPrefix := 'PeerToPeerB::' ) ;
	fbPeerToPeer_1		: FB_PeerToPeer_1;
	fbPeerToPeer_2		: FB_PeerToPeer_2;
	
   	fbTx				: FB_FrameFifo;
	fbTx_1				: FB_FrameFifo_1;
	fbTx_2				: FB_FrameFifo_2;
		
   	fbRx				: FB_FrameFiforx;
	fbLog				: FB_LogFifo;
	  
	stSendTo			: ST_FrameFifoEntrydata;	
	stSendTo_1			: ST_FrameFifoEntrydata_1;
	stSendTo_2			: ST_FrameFifoEntrydata_2;
	
	stReceivedFrom		: ST_FrameFifoEntrydatarx;
	
	sLoggedMessage		: T_MaxString;

   	fbCloseAll 			: FB_SocketCloseAll;
   	bInitialize			: BOOL := TRUE;
	
	
	senddataheader1 : ARRAY[0..11] OF BYTE;
	senddata1 : ARRAY[0..47] OF BYTE;
	
	senddataheader2 : ARRAY[0..11] OF BYTE;
	senddata2 : ARRAY[0..11] OF BYTE;
	
	senddataheader3 : ARRAY[0..11] OF BYTE;
	senddata3 : ARRAY[0..5] OF BYTE;
	
	senddataheader4 : ARRAY[0..12] OF BYTE;
	
	senddataheader5 : ARRAY[0..11] OF BYTE;
	senddata5 : ARRAY[0..3] OF BYTE;
	
	senddataheader6 : ARRAY[0..11] OF BYTE;
	senddata6 : ARRAY[0..3] OF BYTE;
	
	senddataheader7 : ARRAY[0..11] OF BYTE;
	senddata7 : ARRAY[0..3] OF BYTE;
	
	senddataheader8 : ARRAY[0..11] OF BYTE;
	senddata8 : ARRAY[0..3] OF BYTE;
		
	i : INT;	
	udpsendclock : TON;
			
	// made
	
	packetheader1 : ARRAY[0..11] OF BYTE;
	packetdata1 : ARRAY[0..47] OF BYTE;	
	
	packetheader2 : ARRAY[0..11] OF BYTE;
	packetdata2 : ARRAY[0..11] OF  BYTE;
		
	packetheader3 : ARRAY[0..11] OF BYTE;
	packetdata3 : ARRAY[0..5] OF BYTE;
		
	packetheader4 : ARRAY[0..12] OF BYTE;
	diagrst : BYTE;
	
	packetheader5 : ARRAY[0..11] OF BYTE;
	packetdata5 : ARRAY[0..3] OF BYTE;
	
	packetheader6 : ARRAY[0..11] OF BYTE;
	packetdata6 : ARRAY[0..3] OF BYTE;
	
	packetheader7 : ARRAY[0..11] OF BYTE;
	packetdata7 : ARRAY[0..3] OF BYTE;
	
	packetheader8 : ARRAY[0..11] OF BYTE;
	packetdata8 : ARRAY[0..3] OF BYTE;
	

	packetswitch1 : BOOL := FALSE;
	packetswitch2 : BOOL := FALSE;
	packetswitch3 : BOOL := FALSE; // Trigger 5678
	
	
	packetswitch5 : BOOL;
	packetswitch6 : BOOL;
	packetswitch7 : BOOL;
	packetswitch8 : BOOL;
			
	idvalue1 : UINT := 16#0001;
	idvalue2 : UINT := 16#0002;
	idvalue3 : UINT := 16#0003;
	idvalue4 : UINT := 16#0004;
	idvalue5 : UINT := 16#0101;
	idvalue6 : UINT := 16#0102;
	idvalue7 : UINT := 16#0103;
	idvalue8 : UINT := 16#0104;
		
	id1 :  Union_UINT;
	id2 :  Union_UINT;
	id3 :  Union_UINT;
	id4 :  Union_UINT;
	id5 :  Union_UINT;
	id6 :  Union_UINT;
	id7 :  Union_UINT;
	id8 :  Union_UINT;
	
	datalen1 : Union_UDINT;
	datalen2 : Union_UDINT;
	datalen3 : Union_UDINT;
	datalen4 : Union_UDINT;
	datalen5 : Union_UDINT;
	datalen6 : Union_UDINT;
	datalen7 : Union_UDINT;
	datalen8 : Union_UDINT;
	
	txcounter1 : Union_UDINT;
	txcounter2 : Union_UDINT;
	txcounter3 : Union_UDINT;
    txcounter4 : Union_UDINT;
	txcounter5 : Union_UDINT;
	txcounter6 : Union_UDINT;
	txcounter7 : Union_UDINT;
	txcounter8 : Union_UDINT;
	
	rxcounter1 : Union_UDINT;
	rxcounter2 : Union_UDINT;
	rxcounter3 : Union_UDINT;
	rxcounter4 : Union_UDINT;
		
	counter1 : UDINT :=0;
	counter2 : UDINT :=0;
	counter3 : UDINT :=0;
	counter4, counter5, counter6, counter7, counter8 : UDINT :=0; 	
		
	counterreset : BOOL := FALSE;
	
	mcsmission :Union_UINT; // rx	
	mcstarget : Union_UINT; //rx
	runningtime : UDINT ; 
	runningtimetimer : TON;
	targetVelocity : STRING; 	
	errorcheckid : BYTE;
	emgrcmd : BYTE;
	
	packetmcsmission :Union_UINT;    
	packetmcstargetnum : Union_UINT;	
	
	packetmcstarget : Union_UINT;
	packetwetpointlat : Union_LREAL;
	packetwetpointlot : Union_LREAL;
	packetwetpointspeed : Union_REAL;
	
	packetmcstarget1 : Union_UINT;
	packetwetpointlat1 : Union_LREAL;
	packetwetpointlot1 : Union_LREAL;
	packetwetpointspeed1 : Union_UDINT;
	
	packetwetpointlat1str : STRING;
	packetwetpointlot1str : STRING;

	packetmcstarget2 : Union_UINT;
	packetwetpointlat2 : Union_LREAL;	
	packetwetpointlot2 : Union_LREAL;	
	
	packetwetpointspeed2 : Union_UDINT;
	
	packetwetpointlat2str : STRING;
	packetwetpointlot2str : STRING;
		
	packetmcstarget3 : Union_UINT;
	packetwetpointlat3 : Union_LREAL;	
	packetwetpointlot3 : Union_LREAL;
	
	packetwetpointspeed3 : Union_UDINT;
	
	packetwetpointlat3str : STRING;
	packetwetpointlot3str : STRING;
	
	packetmcstarget4 : Union_UINT;
	packetwetpointlat4 : Union_LREAL;	
	packetwetpointlot4 : Union_LREAL;	
	packetwetpointspeed4 : Union_UDINT;
	
	packetmcstarget5,packetmcstarget6,packetmcstarget7,packetmcstarget8,
    packetmcstarget9,packetmcstarget10,packetmcstarget11,packetmcstarget12,packetmcstarget13,
    packetmcstarget14,packetmcstarget15,packetmcstarget16 : Union_UINT;
	
	packetwetpointlat5,packetwetpointlat6,packetwetpointlat7,packetwetpointlat8,
    packetwetpointlat9,packetwetpointlat10,packetwetpointlat11,packetwetpointlat12,packetwetpointlat13,
    packetwetpointlat14,packetwetpointlat15,packetwetpointlat16 : Union_LREAL;
	
	packetwetpointlot5,packetwetpointlot6,packetwetpointlot7,packetwetpointlot8,
    packetwetpointlot9,packetwetpointlot10,packetwetpointlot11,packetwetpointlot12,packetwetpointlot13,
    packetwetpointlot14,packetwetpointlot15,packetwetpointlot16 : Union_LREAL;	
	
	packetwetpointspeed5,packetwetpointspeed6,packetwetpointspeed7,packetwetpointspeed8,
    packetwetpointspeed9,packetwetpointspeed10,packetwetpointspeed11,packetwetpointspeed12,packetwetpointspeed13,
    packetwetpointspeed14,packetwetpointspeed15,packetwetpointspeed16 : Union_UDINT;

	
	packetahrsheading : Union_LREAL;
	packetahrspitch : Union_LREAL;
	packetahrsroll : Union_LREAL;
	packetspeed : Union_LREAL;
	packetlat : Union_LREAL;
	packetlon : Union_LREAL;	
	packetrunningtime : Union_UDINT;
	packetheading : Union_UINT;
	packetvelocity : Union_UINT;
	packetrbbsoc : Union_UINT;
	packetthrusterrightrpm : Union_UINT;
	packetthrusterleftrpm : Union_UINT;	
	packetmissioncmd : Union_UINT;

	emergencydata : BYTE;		 
	controlshutdown : BOOL;
	
END_VAR

VAR_INPUT
	Algorithmtestint : Union_UINT;
	AlgorithmWaypointint : Union_UINT;
	bSendOnceToRemote1	: BOOL := FALSE;(* Rising edge at this variable sends message to the remote host/port *)
	bSendOnceToRemote2	: BOOL := FALSE;(* Rising edge at this variable sends message to the remote host/port *)
	UDPstart : BOOL := TRUE;
	UDPstart2 : BOOL := FALSE;
	UDPstart3 : BOOL := FALSE;
END_VAR
VAR_OUTPUT
	Algorithm_Sw : BOOL := FALSE;
	Algorithmstop : BOOL :=TRUE;
	Receiveaddress : BYTE;
END_VAR


IF UDPstart THEN
fbCloseAll( sSrvNetId := sSrvNetId, bExecute:= bInitialize );
IF fbCloseAll.bBusy OR fbCloseAll.bError THEN
	RETURN;
END_IF
bInitialize := FALSE;

fbPeerToPeer(  sSrvNetId := sSrvNetId, 
				fbTx := fbTx, 
				fbRx := fbRx,			
				fbLog := fbLog, 
				sLocalHost := sLocalHost, 
				nLocalPort := nLocalPort, 
				bEnable := bEnable, bLog := bLog );
																
IF fbPeerToPeer.bCreated  THEN 
	
// Receive Control
Receiveaddress := stReceivedFrom.rxdata[2]; 

IF Receiveaddress = 16#01 THEN 
	
   mcsmission.packed[0] := stReceivedFrom.rxdata[12]; 
   mcsmission.packed[1] := stReceivedFrom.rxdata[13];
   	  
END_IF 

IF Receiveaddress = 16#02 THEN 
		
	packetmcstargetnum.packed[0] := stReceivedFrom.rxdata[12]; //12
    packetmcstargetnum.packed[1] := stReceivedFrom.rxdata[13];
	
	packetmcstarget1.packed[0] :=  stReceivedFrom.rxdata[14];
	packetmcstarget1.packed[1] :=  stReceivedFrom.rxdata[15];
	
	FOR i:=0 TO 7 BY 1 DO
	packetwetpointlat1.packed[i] :=  stReceivedFrom.rxdata[i+16];
	END_FOR
	FOR i:=0 TO 7 BY 1 DO
	packetwetpointlot1.packed[i] :=  stReceivedFrom.rxdata[i+24];
	END_FOR	
	FOR i:=0 TO 3 BY 1 DO
	packetwetpointspeed1.packed[i] :=  stReceivedFrom.rxdata[i+32];
	END_FOR
	
	packetmcstarget2.packed[0] :=  stReceivedFrom.rxdata[36];
	packetmcstarget2.packed[1] :=  stReceivedFrom.rxdata[37];
	
	FOR i:=0 TO 7 BY 1 DO
	packetwetpointlat2.packed[i] :=  stReceivedFrom.rxdata[i+38];
	END_FOR
	FOR i:=0 TO 7 BY 1 DO
	packetwetpointlot2.packed[i] :=  stReceivedFrom.rxdata[i+46];
	END_FOR
	FOR i:=0 TO 3 BY 1 DO
	packetwetpointspeed2.packed[i] :=  stReceivedFrom.rxdata[i+54];
	END_FOR
		
	packetmcstarget3.packed[0] :=  stReceivedFrom.rxdata[58];
	packetmcstarget3.packed[1] :=  stReceivedFrom.rxdata[59];
	
	FOR i:=0 TO 7 BY 1 DO
	packetwetpointlat3.packed[i] := stReceivedFrom.rxdata[i+60];
	END_FOR
	FOR i:=0 TO 7 BY 1 DO
	packetwetpointlot3.packed[i] :=  stReceivedFrom.rxdata[i+68];
	END_FOR
	FOR i:=0 TO 3 BY 1 DO
	packetwetpointspeed3.packed[i] :=  stReceivedFrom.rxdata[i+76];
	END_FOR
	
	packetmcstarget4.packed[0] :=  stReceivedFrom.rxdata[80];
	packetmcstarget4.packed[1] := stReceivedFrom.rxdata[81];
	
	FOR i:=0 TO 7 BY 1 DO
	packetwetpointlat4.packed[i] :=  stReceivedFrom.rxdata[i+82];
	END_FOR
	FOR i:=0 TO 7 BY 1 DO
	packetwetpointlot4.packed[i] :=  stReceivedFrom.rxdata[i+90];
	END_FOR
	FOR i:=0 TO 3 BY 1 DO
	packetwetpointspeed4.packed[i] :=  stReceivedFrom.rxdata[i+98];
	END_FOR	
		
	packetmcstarget5.packed[0] :=  stReceivedFrom.rxdata[102];
	packetmcstarget5.packed[1] := stReceivedFrom.rxdata[103];
	
	FOR i:=0 TO 7 BY 1 DO
	packetwetpointlat5.packed[i] :=  stReceivedFrom.rxdata[i+104];
	END_FOR
	FOR i:=0 TO 7 BY 1 DO
	packetwetpointlot5.packed[i] :=  stReceivedFrom.rxdata[i+112];
	END_FOR
	FOR i:=0 TO 3 BY 1 DO
	packetwetpointspeed5.packed[i] :=  stReceivedFrom.rxdata[i+120];
	END_FOR	
	
	packetmcstarget6.packed[0] :=  stReceivedFrom.rxdata[124];
	packetmcstarget6.packed[1] := stReceivedFrom.rxdata[125];
	
	FOR i:=0 TO 7 BY 1 DO
	packetwetpointlat6.packed[i] :=  stReceivedFrom.rxdata[i+126];
	END_FOR
	FOR i:=0 TO 7 BY 1 DO
	packetwetpointlot6.packed[i] :=  stReceivedFrom.rxdata[i+134];
	END_FOR
	FOR i:=0 TO 3 BY 1 DO
	packetwetpointspeed6.packed[i] :=  stReceivedFrom.rxdata[i+142];
	END_FOR	
	
	packetmcstarget7.packed[0] :=  stReceivedFrom.rxdata[146];
	packetmcstarget7.packed[1] := stReceivedFrom.rxdata[147];
	
	FOR i:=0 TO 7 BY 1 DO
	packetwetpointlat7.packed[i] :=  stReceivedFrom.rxdata[i+148];
	END_FOR
	FOR i:=0 TO 7 BY 1 DO
	packetwetpointlot7.packed[i] :=  stReceivedFrom.rxdata[i+156];
	END_FOR
	FOR i:=0 TO 3 BY 1 DO
	packetwetpointspeed7.packed[i] :=  stReceivedFrom.rxdata[i+164];
	END_FOR	
	
	packetmcstarget8.packed[0] :=  stReceivedFrom.rxdata[168];
	packetmcstarget8.packed[1] := stReceivedFrom.rxdata[169];
	
	FOR i:=0 TO 7 BY 1 DO
	packetwetpointlat8.packed[i] :=  stReceivedFrom.rxdata[i+170];
	END_FOR
	FOR i:=0 TO 7 BY 1 DO
	packetwetpointlot8.packed[i] :=  stReceivedFrom.rxdata[i+178];
	END_FOR
	FOR i:=0 TO 3 BY 1 DO
	packetwetpointspeed8.packed[i] :=  stReceivedFrom.rxdata[i+186];
	END_FOR	
	
	packetmcstarget9.packed[0] :=  stReceivedFrom.rxdata[190];
	packetmcstarget9.packed[1] := stReceivedFrom.rxdata[191];
	
	FOR i:=0 TO 7 BY 1 DO
	packetwetpointlat9.packed[i] :=  stReceivedFrom.rxdata[i+192];
	END_FOR
	FOR i:=0 TO 7 BY 1 DO
	packetwetpointlot9.packed[i] :=  stReceivedFrom.rxdata[i+200];
	END_FOR
	FOR i:=0 TO 3 BY 1 DO
	packetwetpointspeed9.packed[i] :=  stReceivedFrom.rxdata[i+208];
	END_FOR	
	
	packetmcstarget10.packed[0] :=  stReceivedFrom.rxdata[212];
	packetmcstarget10.packed[1] := stReceivedFrom.rxdata[213];
	
	FOR i:=0 TO 7 BY 1 DO
	packetwetpointlat10.packed[i] :=  stReceivedFrom.rxdata[i+214];
	END_FOR
	FOR i:=0 TO 7 BY 1 DO
	packetwetpointlot10.packed[i] :=  stReceivedFrom.rxdata[i+222];
	END_FOR
	FOR i:=0 TO 3 BY 1 DO
	packetwetpointspeed10.packed[i] :=  stReceivedFrom.rxdata[i+230];
	END_FOR	
	
	packetmcstarget11.packed[0] :=  stReceivedFrom.rxdata[234];
	packetmcstarget11.packed[1] := stReceivedFrom.rxdata[235];
	
	FOR i:=0 TO 7 BY 1 DO
	packetwetpointlat11.packed[i] :=  stReceivedFrom.rxdata[i+236];
	END_FOR
	FOR i:=0 TO 7 BY 1 DO
	packetwetpointlot11.packed[i] :=  stReceivedFrom.rxdata[i+244];
	END_FOR
	FOR i:=0 TO 3 BY 1 DO
	packetwetpointspeed11.packed[i] :=  stReceivedFrom.rxdata[i+252];
	END_FOR	
	
	packetmcstarget12.packed[0] :=  stReceivedFrom.rxdata[256];
	packetmcstarget12.packed[1] := stReceivedFrom.rxdata[257];
	
	FOR i:=0 TO 7 BY 1 DO
	packetwetpointlat12.packed[i] :=  stReceivedFrom.rxdata[i+258];
	END_FOR
	FOR i:=0 TO 7 BY 1 DO
	packetwetpointlot12.packed[i] :=  stReceivedFrom.rxdata[i+266];
	END_FOR
	FOR i:=0 TO 3 BY 1 DO
	packetwetpointspeed12.packed[i] :=  stReceivedFrom.rxdata[i+274];
	END_FOR	
	
	packetmcstarget13.packed[0] :=  stReceivedFrom.rxdata[278];
	packetmcstarget13.packed[1] := stReceivedFrom.rxdata[279];
	
	FOR i:=0 TO 7 BY 1 DO
	packetwetpointlat13.packed[i] :=  stReceivedFrom.rxdata[i+280];
	END_FOR
	FOR i:=0 TO 7 BY 1 DO
	packetwetpointlot13.packed[i] :=  stReceivedFrom.rxdata[i+288];
	END_FOR
	FOR i:=0 TO 3 BY 1 DO
	packetwetpointspeed13.packed[i] :=  stReceivedFrom.rxdata[i+296];
	END_FOR	
	
	packetmcstarget14.packed[0] :=  stReceivedFrom.rxdata[300];
	packetmcstarget14.packed[1] := stReceivedFrom.rxdata[301];
	
	FOR i:=0 TO 7 BY 1 DO
	packetwetpointlat14.packed[i] :=  stReceivedFrom.rxdata[i+302];
	END_FOR
	FOR i:=0 TO 7 BY 1 DO
	packetwetpointlot14.packed[i] :=  stReceivedFrom.rxdata[i+310];
	END_FOR
	FOR i:=0 TO 3 BY 1 DO
	packetwetpointspeed14.packed[i] :=  stReceivedFrom.rxdata[i+318];
	END_FOR	
	
	packetmcstarget15.packed[0] :=  stReceivedFrom.rxdata[322];
	packetmcstarget15.packed[1] := stReceivedFrom.rxdata[323];
	
	FOR i:=0 TO 7 BY 1 DO
	packetwetpointlat15.packed[i] :=  stReceivedFrom.rxdata[i+324];
	END_FOR
	FOR i:=0 TO 7 BY 1 DO
	packetwetpointlot15.packed[i] :=  stReceivedFrom.rxdata[i+332];
	END_FOR
	FOR i:=0 TO 3 BY 1 DO
	packetwetpointspeed15.packed[i] :=  stReceivedFrom.rxdata[i+340];
	END_FOR	
	
	packetmcstarget16.packed[0] :=  stReceivedFrom.rxdata[344];
	packetmcstarget16.packed[1] := stReceivedFrom.rxdata[345];
	
	FOR i:=0 TO 7 BY 1 DO
	packetwetpointlat16.packed[i] :=  stReceivedFrom.rxdata[i+346];
	END_FOR
	FOR i:=0 TO 7 BY 1 DO
	packetwetpointlot16.packed[i] :=  stReceivedFrom.rxdata[i+354];
	END_FOR
	FOR i:=0 TO 3 BY 1 DO
	packetwetpointspeed16.packed[i] :=  stReceivedFrom.rxdata[i+362];
	END_FOR	
	 
END_IF 
(*IF Receiveaddress = 16#03 THEN 
	
END_IF*)

IF Receiveaddress = 16#04THEN 
	emergencydata := stReceivedFrom.rxdata[12];  
END_IF 


// UDP_1 1HZ trigger 
udpsendclock(IN:=TRUE, PT:=T#1S); //T#1S

 IF udpsendclock.Q THEN
    bSendOnceToRemote := NOT bSendOnceToRemote;
    udpsendclock(IN:=FALSE);
 END_IF 

// UDP_1 Send Packet Control

IF bSendOnceToRemote THEN
     bSendOnceToRemote 	         := TRUE;		
	 stSendTo.stRemoteAddr.sAddr := sRemoteHost;	
	 stSendTo.stRemoteAddr.nPort := nRemotePort;

IF counterreset THEN
	counter1 :=0;
	counter2 :=0;
	counter3 :=0;
 END_IF 

counter1 := counter1+1;
counter2 := counter2+1;
counter3 := counter3+1;

id1.value := idvalue1;
id2.value := idvalue2;
id3.value := idvalue3;

datalen1.value := SIZEOF(packetdata1);
datalen2.value := SIZEOF(packetdata2);
datalen3.value := SIZEOF(packetdata3);

txcounter1.value := counter1;
txcounter2.value := counter2;
txcounter3.value := counter3;

packetwetpointspeed.value := 1.082;
targetVelocity := REAL_TO_STRING(packetwetpointspeed.value); // target

packetahrsheading.value :=STRING_TO_LREAL(MAIN.HMIYAW);
packetahrspitch.value := STRING_TO_LREAL(MAIN.HMIPITCH);
packetahrsroll.value := STRING_TO_LREAL(MAIN.HMIROLL);
packetlat.value := STRING_TO_LREAL(MAIN.HMILatitude);
packetlon.value := STRING_TO_LREAL(MAIN.HMILongitude);
packetspeed.value := STRING_TO_LREAL(MAIN.HMISpeed);

packetrunningtime.value := runningtime;
packetheading.value := LREAL_TO_UINT(MAIN.azimuth);
packetvelocity.value := STRING_TO_UINT(targetvelocity);

packetrbbsoc.value := STRING_TO_UINT(MAIN.HMIbatS);
packetthrusterrightrpm.value := MAIN.thrusterrightrpm;
packetthrusterleftrpm.value := MAIN.thrusterleftrpm;
packetmcstarget.value := MAIN.waypointIndex;

 IF mcsmission.value = 1 THEN // rx
	  packetmcsmission.value :=1; // tx
	  Algorithm_Sw := TRUE;
	  runningtimetimer(IN:=TRUE,PT:=T#1S);
         IF runningtimetimer.Q THEN
	        runningtime := runningtime+1;
	        runningtimetimer(IN:=FALSE);
         END_IF
      ELSIF mcsmission.value = 2 THEN
		packetmcsmission.value :=0;
		runningtime :=0;
		Algorithmstop := FALSE;
	  ELSIF mcsmission.value = 3 THEN
		packetmcsmission.value :=2;  
		Algorithm_Sw := FALSE;
		runningtimetimer(IN:=TRUE,PT:=T#1S);
         IF runningtimetimer.Q THEN
	        runningtime := runningtime+1;
	        runningtimetimer(IN:=FALSE);
         END_IF
	   ELSIF mcsmission.value = 4 THEN
		   controlshutdown := TRUE;
END_IF 

IF emergencydata = 16#02 THEN
   packetmcsmission.value :=0;
   runningtime :=0;
   Algorithmstop := FALSE;
   ELSIF emergencydata = 16#01 THEN
	    Algorithmstop := TRUE;
		packetmcsmission.value :=1;
		runningtimetimer(IN:=TRUE,PT:=T#1S);
         IF runningtimetimer.Q THEN
	        runningtime := runningtime+1;
	        runningtimetimer(IN:=FALSE);
         END_IF
END_IF


// UDP_1 packet1 

packetheader1[0] := 16#30;
packetheader1[1] := 16#10;

packetheader1[2] := id1.packed[0];
packetheader1[3] := id1.packed[1];
FOR i:=0 TO 3 BY 1 DO
packetheader1[i+4] := datalen1.packed[i];
END_FOR
FOR i:=0 TO 3 BY 1 DO
packetheader1[i+8] := txcounter1.packed[i];
END_FOR
FOR i:=0 TO 7 BY 1 DO
packetdata1[i] := packetahrsroll.Packed[i];	
END_FOR
FOR i:=0 TO 7 BY 1 DO
packetdata1[i+8] := packetahrspitch.Packed[i];	
END_FOR
FOR i:=0 TO 7 BY 1 DO
packetdata1[i+16] := packetahrsheading.Packed[i];	
END_FOR
FOR i:=0 TO 7 BY 1 DO
packetdata1[i+24] := packetspeed.Packed[i];	
END_FOR
FOR i:=0 TO 7 BY 1 DO
packetdata1[i+32] := packetlat.Packed[i];	
END_FOR
FOR i:=0 TO 7 BY 1 DO
packetdata1[i+40] := packetlon.Packed[i];	
END_FOR


// UDP_1 packet2

packetheader2[0] := 16#30;
packetheader2[1] := 16#10;

packetheader2[2] := id2.packed[0];
packetheader2[3] := id2.packed[1];
FOR i:=0 TO 3 BY 1 DO
packetheader2[i+4] := datalen2.packed[i];
END_FOR
FOR i:=0 TO 3 BY 1 DO
packetheader2[i+8] := txcounter2.packed[i];
END_FOR

packetdata2[0] := packetmcsmission.packed[0];
packetdata2[1] := packetmcsmission.packed[1];

packetdata2[2] :=  packetmcstarget.packed[0];
packetdata2[3] :=  packetmcstarget.packed[1];

packetdata2[4] := packetrunningtime.packed[0];
packetdata2[5] := packetrunningtime.packed[1];
packetdata2[6] := packetrunningtime.packed[2];
packetdata2[7] := packetrunningtime.packed[3];

packetdata2[8] := packetheading.packed[0];  // GPS 
packetdata2[9] := packetheading.packed[1];

packetdata2[10] := packetvelocity.packed[0]; // 2KNOT
packetdata2[11] := packetvelocity.packed[1];

// UDP_1 packet3

packetheader3[0] := 16#30;

packetheader3[1] := 16#10;

packetheader3[2] := id3.packed[0];
packetheader3[3] := id3.packed[1];
FOR i:=0 TO 3 BY 1 DO
packetheader3[i+4] := datalen3.packed[i];
END_FOR
FOR i:=0 TO 3 BY 1 DO
packetheader3[i+8] := txcounter3.packed[i];
END_FOR

packetdata3[0] := packetrbbsoc.packed[0];
packetdata3[1] := packetrbbsoc.packed[1];

packetdata3[2] := packetthrusterrightrpm.packed[0];
packetdata3[3] := packetthrusterrightrpm.packed[1];

packetdata3[4] := packetthrusterleftrpm.packed[0];
packetdata3[5] := packetthrusterleftrpm.packed[1];

// UDP_1 Packet1 Send	
        FOR i:=0 TO 11 BY 1 DO
			senddataheader1[i] := packetheader1[i];
		END_FOR
		FOR i:=0 TO 47 BY 1 DO
			senddata1[i] := packetdata1[i];
		END_FOR
		FOR i:=0 TO 11 BY 1 DO
			stSendTO.txdata[i] := senddataheader1[i];
		END_FOR
		FOR i:=0 TO 47 BY 1 DO
			stSendTO.txdata[i+12] := senddata1[i];
		END_FOR 
// UDP_1 Packet2 Send			
		FOR i:=0 TO 11 BY 1 DO
			senddataheader2[i] := packetheader2[i];
		END_FOR
		FOR i:=0 TO 11 BY 1 DO
			senddata2[i] := packetdata2[i];
		END_FOR		
		FOR i:=0 TO 11 BY 1 DO
			stSendTO.txdata[i+60] := senddataheader2[i];
		END_FOR
		FOR i:=0 TO 11 BY 1 DO
			stSendTO.txdata[i+72] := senddata2[i];
		END_FOR		
// UDP_1 Packet3 Send	
		FOR i:=0 TO 11 BY 1 DO
			senddataheader3[i] := packetheader3[i];
		END_FOR
		FOR i:=0 TO 5 BY 1 DO
			senddata3[i] := packetdata3[i];
		END_FOR		
		FOR i:=0 TO 11 BY 1 DO
			stSendTO.txdata[i+84] := senddataheader3[i];
		END_FOR
		FOR i:=0 TO 5 BY 1 DO
			stSendTO.txdata[i+96] := senddata3[i];
		END_FOR  
	 
	 fbTx.AddTail( stPut := stSendTo); // UDP_1 send
	IF NOT fbTx.bOk THEN				
			fbLog.Error( sMessage := 'FB_FrameFifo(sender)', nErrID := PLCPRJ_ERROR_SENDFIFO_OVERFLOW );
		END_IF		
END_IF

	IF bSendOnceToRemote THEN
	bSendOnceToRemote := FALSE;
	END_IF  
		
END_IF

REPEAT
	fbRx.RemoveHead();
	IF fbRx.bOk THEN
	stReceivedFrom := fbRx.stGet;		
	END_IF
UNTIL NOT fbRx.bOk
END_REPEAT

REPEAT
	fbLog.Remove( );
	IF fbLog.bOk THEN
		sLoggedMessage := fbLog.sGet;
	END_IF
UNTIL NOT fbLog.bOk
END_REPEAT
ELSE 
	
fbPeerToPeer(   sSrvNetId := sSrvNetId, 
				fbTx := fbTx, 
				fbRx := fbRx,			
				fbLog := fbLog, 
				sLocalHost := sLocalHost, 
				nLocalPort := nLocalPort, 
				bEnable := FALSE, bLog := bLog );
END_IF

// Namespace : UDP_2

IF UDPstart2 THEN	
fbCloseAll( sSrvNetId := sSrvNetId, bExecute:= bInitialize );
IF fbCloseAll.bBusy OR fbCloseAll.bError THEN
	RETURN;
END_IF
bInitialize := FALSE;

fbPeerToPeer_1(  sSrvNetId := sSrvNetId, 
				fbTx := fbTx_1, 
				fbRx := fbRx,			
				fbLog := fbLog, 
				sLocalHost := sLocalHost, 
				nLocalPort := nLocalPort, 
				bEnable := bEnable, bLog := bLog );

IF fbPeerToPeer_1.bCreated THEN 

ReceiveAddress := stReceivedFrom.rxdata[2]; 	
// UDP_2 Send Packet Control

IF NOT bSendOnceToRemote1 THEN	
	 stSendTo_1.stRemoteAddr.sAddr := sRemoteHost;	
	 stSendTo_1.stRemoteAddr.nPort := nRemotePort;

IF counterreset THEN
	counter4 :=0;
 END_IF 

counter4 := counter4+1;

id4.value := idvalue4;

datalen4.value := SIZEOF(diagrst);

txcounter4.value := counter4;

packetahrsheading.value :=STRING_TO_LREAL(MAIN.HMIYAW);
packetlat.value := STRING_TO_LREAL(MAIN.HMILatitude);
packetlon.value := STRING_TO_LREAL(MAIN.HMILongitude);

IF packetahrsheading.value =0 AND packetlat.value =0 AND packetlon.value=0 THEN
	diagrst := 0;
	ELSE
		diagrst := 16#01;
	END_IF
	
// UDP_2 packet4 

packetheader4[0] := 16#30;

packetheader4[1] := 16#10;

packetheader4[2] := id4.packed[0];
packetheader4[3] := id4.packed[1];

packetheader4[4] := datalen4.packed[0];
packetheader4[5] := datalen4.packed[1];
packetheader4[6] := datalen4.packed[2];
packetheader4[7] := datalen4.packed[3];

packetheader4[8] := txcounter4.packed[0];
packetheader4[9] := txcounter4.packed[1];
packetheader4[10] := txcounter4.packed[2];
packetheader4[11] := txcounter4.packed[3];

packetheader4[12] := diagrst;


// UDP_2 Packet4 Send	
    	FOR i:=0 TO 12 BY 1 DO
			senddataheader4[i] := packetheader4[i];
		END_FOR		
		FOR i:=0 TO 12 BY 1 DO
			stSendTO_1.txdata[i] := senddataheader4[i];
		END_FOR
	 
	 fbTx_1.AddTail( stPut := stSendTo_1);// UDP_2 send
	IF NOT fbTx_1.bOk THEN				
			fbLog.Error( sMessage := 'FB_FrameFifo(sender)', nErrID := PLCPRJ_ERROR_SENDFIFO_OVERFLOW );
		END_IF		
END_IF

	IF NOT bSendOnceToRemote1 THEN
	bSendOnceToRemote1 := TRUE;
	END_IF  
		
END_IF

REPEAT
	fbRx.RemoveHead();
	IF fbRx.bOk THEN
	stReceivedFrom := fbRx.stGet;		
	END_IF
UNTIL NOT fbRx.bOk
END_REPEAT

REPEAT
	fbLog.Remove( );
	IF fbLog.bOk THEN
		sLoggedMessage := fbLog.sGet;
	END_IF
UNTIL NOT fbLog.bOk
END_REPEAT

ELSE 

fbPeerToPeer_1( sSrvNetId := sSrvNetId, 
				fbTx := fbTx_1, 
				fbRx := fbRx,			
				fbLog := fbLog, 
				sLocalHost := sLocalHost, 
				nLocalPort := nLocalPort, 
				bEnable := FALSE, bLog := bLog );


END_IF

IF UDPstart3 THEN
	
fbCloseAll( sSrvNetId := sSrvNetId, bExecute:= bInitialize );
IF fbCloseAll.bBusy OR fbCloseAll.bError THEN
	RETURN;
END_IF
bInitialize := FALSE;

fbPeerToPeer_2(   sSrvNetId := sSrvNetId, 
				fbTx := fbTx_2, 
				fbRx := fbRx,			
				fbLog := fbLog, 
				sLocalHost := sLocalHost, 
				nLocalPort := nLocalPort, 
				bEnable := bEnable, bLog := bLog );

IF fbPeerToPeer_2.bCreated THEN 

// UDP_3 Receive Control
 
Receiveaddress := stReceivedFrom.rxdata[2]; 

IF Receiveaddress = 16#01 THEN
   packetswitch5  := TRUE;	 
  rxcounter1.packed[0] := stReceivedFrom.rxdata[8];
  rxcounter1.packed[1] := stReceivedFrom.rxdata[9];
  rxcounter1.packed[2] := stReceivedFrom.rxdata[10];
  rxcounter1.packed[3] := stReceivedFrom.rxdata[11];
ELSE  packetswitch5  := FALSE;	
END_IF 


IF Receiveaddress = 16#02 THEN
	packetswitch6  := TRUE;		
	rxcounter2.packed[0] := stReceivedFrom.rxdata[8];
    rxcounter2.packed[1] := stReceivedFrom.rxdata[9];
    rxcounter2.packed[2] := stReceivedFrom.rxdata[10];
    rxcounter2.packed[3] := stReceivedFrom.rxdata[11];
ELSE  packetswitch6  := FALSE;	
END_IF

IF Receiveaddress = 16#03 THEN
    packetswitch7  := TRUE;
	rxcounter3.packed[0] := stReceivedFrom.rxdata[8];
    rxcounter3.packed[1] := stReceivedFrom.rxdata[9];
    rxcounter3.packed[2] := stReceivedFrom.rxdata[10];
    rxcounter3.packed[3] := stReceivedFrom.rxdata[11];
ELSE  packetswitch7  := FALSE;	
END_IF

IF Receiveaddress = 16#04 THEN
    packetswitch8  := TRUE;
	rxcounter4.packed[0] := stReceivedFrom.rxdata[8];
    rxcounter4.packed[1] := stReceivedFrom.rxdata[9];
    rxcounter4.packed[2] := stReceivedFrom.rxdata[10];
    rxcounter4.packed[3] := stReceivedFrom.rxdata[11];
ELSE  packetswitch8  := FALSE;	
END_IF

// UDP_3 Send Packet Control

IF NOT bSendOnceToRemote2 THEN	
	 stSendTo_2.stRemoteAddr.sAddr := sRemoteHost;	
	 stSendTo_2.stRemoteAddr.nPort := nRemotePort;
	 
IF counterreset THEN
	counter5 :=0;
    counter6 :=0;
    counter7 :=0;
    counter8 :=0;
 END_IF 

counter5 := counter5+1;
counter6 := counter6+1;
counter7 := counter7+1;
counter8 := counter8+1;

id5.value := idvalue5;
id6.value := idvalue6;
id7.value := idvalue7;
id8.value := idvalue8;

datalen5.value := SIZEOF(packetdata5);
datalen6.value := SIZEOF(packetdata6);
datalen7.value := SIZEOF(packetdata7);
datalen8.value := SIZEOF(packetdata8);

txcounter5.value := counter5;
txcounter6.value := counter6;
txcounter7.value := counter7;
txcounter8.value := counter8;

// UDP_3 packet5

packetheader5[0] := 16#30;

packetheader5[1] := 16#10;

packetheader5[2] := id5.packed[0];
packetheader5[3] := id5.packed[1];

packetheader5[4] := datalen5.packed[0];
packetheader5[5] := datalen5.packed[1];
packetheader5[6] := datalen5.packed[2];
packetheader5[7] := datalen5.packed[3];

packetheader5[8] := txcounter5.packed[0];
packetheader5[9] := txcounter5.packed[1];
packetheader5[10] := txcounter5.packed[2];
packetheader5[11] := txcounter5.packed[3];

packetdata5[0] := rxcounter1.packed[0];
packetdata5[1] := rxcounter1.packed[1];
packetdata5[2] := rxcounter1.packed[2];
packetdata5[3] := rxcounter1.packed[3];

// UDP_3 packet6

packetheader6[0] := 16#30;

packetheader6[1] := 16#10;

packetheader6[2] := id6.packed[0];
packetheader6[3] := id6.packed[1];

packetheader6[4] := datalen6.packed[0];
packetheader6[5] := datalen6.packed[1];
packetheader6[6] := datalen6.packed[2];
packetheader6[7] := datalen6.packed[3];

packetheader6[8] := txcounter6.packed[0];
packetheader6[9] := txcounter6.packed[1];
packetheader6[10] := txcounter6.packed[2];
packetheader6[11] := txcounter6.packed[3];

packetdata6[0] := rxcounter2.packed[0];
packetdata6[1] := rxcounter2.packed[1];
packetdata6[2] := rxcounter2.packed[2];
packetdata6[3] := rxcounter2.packed[3];

// UDP_3 packet7

packetheader7[0] := 16#30;

packetheader7[1] := 16#10;

packetheader7[2] := id7.packed[0];
packetheader7[3] := id7.packed[1];

packetheader7[4] := datalen7.packed[0];
packetheader7[5] := datalen7.packed[1];
packetheader7[6] := datalen7.packed[2];
packetheader7[7] := datalen7.packed[3];

packetheader7[8] := txcounter7.packed[0];
packetheader7[9] := txcounter7.packed[1];
packetheader7[10] := txcounter7.packed[2];
packetheader7[11] := txcounter7.packed[3];

packetdata7[0] := rxcounter3.packed[0];
packetdata7[1] := rxcounter3.packed[1];
packetdata7[2] := rxcounter3.packed[2];
packetdata7[3] := rxcounter3.packed[3];


// UDP_3 packet8

packetheader8[0] := 16#30;

packetheader8[1] := 16#10;

packetheader8[2] := id8.packed[0];
packetheader8[3] := id8.packed[1];

packetheader8[4] := datalen8.packed[0];
packetheader8[5] := datalen8.packed[1];
packetheader8[6] := datalen8.packed[2];
packetheader8[7] := datalen8.packed[3];

packetheader8[8] := txcounter8.packed[0];
packetheader8[9] := txcounter8.packed[1];
packetheader8[10] := txcounter8.packed[2];
packetheader8[11] := txcounter8.packed[3];

packetdata8[0] := rxcounter4.packed[0];
packetdata8[1] := rxcounter4.packed[1];
packetdata8[2] := rxcounter4.packed[2];
packetdata8[3] := rxcounter4.packed[3];

// UDP_3 Packet5 Send	
IF packetswitch5 THEN
        FOR i:=0 TO 11 BY 1 DO
			senddataheader5[i] := packetheader5[i];
		END_FOR
		FOR i:=0 TO 3 BY 1 DO
			senddata5[i] := packetdata5[i];
		END_FOR		
		FOR i:=0 TO 11 BY 1 DO
			stSendTO_2.txdata[i] := senddataheader5[i];
		END_FOR
		FOR i:=0 TO 3 BY 1 DO
			stSendTO_2.txdata[i+12] := senddata5[i];
		END_FOR

 END_IF
 
// UDP_3 Packet6 Send
 IF packetswitch6 THEN
        FOR i:=0 TO 11 BY 1 DO
			senddataheader6[i] := packetheader6[i];
		END_FOR
		FOR i:=0 TO 3 BY 1 DO
			senddata6[i] := packetdata6[i];
		END_FOR		
		FOR i:=0 TO 11 BY 1 DO
			stSendTO_2.txdata[i] := senddataheader6[i];
		END_FOR
		FOR i:=0 TO 3 BY 1 DO
			stSendTO_2.txdata[i+12] := senddata6[i];
		END_FOR		

 END_IF
 
// UDP_3 Packet7 Send
 IF packetswitch7 THEN
        FOR i:=0 TO 11 BY 1 DO
			senddataheader7[i] := packetheader7[i];
		END_FOR
		FOR i:=0 TO 3 BY 1 DO
			senddata7[i] := packetdata7[i];
		END_FOR		
		FOR i:=0 TO 11 BY 1 DO
			stSendTO_2.txdata[i] := senddataheader7[i];
		END_FOR
		FOR i:=0 TO 3 BY 1 DO
			stSendTO_2.txdata[i+12] := senddata7[i];
		END_FOR	

 END_IF
 
// UDP_3 Packet8 Send
 IF packetswitch8 THEN
        FOR i:=0 TO 11 BY 1 DO
			senddataheader8[i] := packetheader8[i];
		END_FOR
		FOR i:=0 TO 3 BY 1 DO
			senddata8[i] := packetdata8[i];
		END_FOR		
		FOR i:=0 TO 11 BY 1 DO
			stSendTO_2.txdata[i] := senddataheader8[i];
		END_FOR
		FOR i:=0 TO 3 BY 1 DO
			stSendTO_2.txdata[i+12] := senddata8[i];
		END_FOR	

 END_IF		

 
	fbTx_2.AddTail( stPut := stSendTo_2); // UDP_3 send
	IF NOT fbTx_2.bOk THEN				
			fbLog.Error( sMessage := 'FB_FrameFifo(sender)', nErrID := PLCPRJ_ERROR_SENDFIFO_OVERFLOW );
		END_IF		
END_IF
	IF NOT bSendOnceToRemote2 THEN
	bSendOnceToRemote2 := TRUE;
	END_IF  
	
END_IF

REPEAT
	fbRx.RemoveHead();
	IF fbRx.bOk THEN
	stReceivedFrom := fbRx.stGet;		
	END_IF
UNTIL NOT fbRx.bOk
END_REPEAT

REPEAT
	fbLog.Remove( );
	IF fbLog.bOk THEN
		sLoggedMessage := fbLog.sGet;
	END_IF
UNTIL NOT fbLog.bOk
END_REPEAT


ELSE	
	fbPeerToPeer_2( sSrvNetId := sSrvNetId, 
				fbTx := fbTx_2, 
				fbRx := fbRx,			
				fbLog := fbLog, 
				sLocalHost := sLocalHost, 
				nLocalPort := nLocalPort, 
				bEnable := FALSE, bLog := bLog );
END_IF

END_PROGRAM

// ---- POUs/FUCTION BLOCK/UDP Source/FB_PeerToPeer.TcPOU

FUNCTION_BLOCK FB_PeerToPeer
VAR_IN_OUT
	fbTx	    : FB_FrameFifo;
	fbRx		: FB_FrameFiforx;
	fbLog		: FB_LogFifo;
	//bCreated		: BOOL;
END_VAR
VAR_INPUT
	sSrvNetId		: T_AmsNetID 	:= '';
	sLocalHost		: T_IPv4Addr 	:= '192.168.10.30';
	nLocalPort		: UDINT 		:= 53634;
	bEnable 		: BOOL			:= FALSE;
	tReconnect		: TIME			:= T#5S;
	bLog			: BOOL			:= FALSE;
	sPrefix			: STRING 		:= 'PeerToPeerX::';
	
	
END_VAR
VAR_OUTPUT
	bCreated		: BOOL;
END_VAR
VAR
	fbCreate		: FB_SocketUdpCreate;
	fbClose			: FB_SocketClose;
	fbReceiveFrom	: FB_SocketUdpReceiveFrom;
	fbSendTo		: FB_SocketUdpSendTo;
	
	stSendTo		: ST_FrameFifoEntrydata;
	stReceivedFrom	: ST_FrameFifoEntrydatarx;
	
	fbCreateTimer	: TON := ( PT := T#0S );	
	eStep			: E_ClientServerSteps;
	
	reseteventerror : BOOL; 
END_VAR

CASE eStep OF
	eUDP_STATE_IDLE:
		IF bEnable XOR bCreated THEN
			IF bEnable THEN
				fbTx.Clear( stput := stSendTo, bLog := bLog );
				fbRx.Clear( stput := stReceivedFrom, bLog := bLog );
				fbLog.Clear( sPrefix := sPrefix, bLog := bLog );

				fbCreateTimer( IN := TRUE );
				IF fbCreateTimer.Q THEN
					fbCreateTimer( IN := FALSE, PT := tReconnect ); 
					eStep := eUDP_STATE_CREATE_START;
				END_IF
			ELSE
				eStep := eUDP_STATE_CLOSE_START;
			END_IF
		ELSIF bCreated THEN
		fbTx.RemoveHead( stGet => stSendTo );
		IF fbTx.bok THEN
		   eStep := eUDP_STATE_SEND_START;
		ELSE 
		   eStep := eUDP_STATE_RECEIVE_START;
		END_IF
	ELSE
		fbCreateTimer( IN := FALSE, PT := T#0S );
		END_IF

	eUDP_STATE_CREATE_START:
		fbCreate( bExecute := FALSE  );
		fbCreate( sSrvNetId := sSrvNetId, sLocalHost:= sLocalHost, nLocalPort:= nLocalPort, bExecute:= TRUE );
		eStep := eUDP_STATE_CREATE_WAIT;

	eUDP_STATE_CREATE_WAIT:
		fbCreate( bExecute := FALSE );
		IF NOT fbCreate.bBusy THEN
			IF NOT fbCreate.bError THEN
				bCreated := TRUE;
				fbLog.Message( sMessage := 'Connectionless (UDP) socket created!', hSocket := fbCreate.hSocket );
				eStep := eUDP_STATE_IDLE;
			ELSE
				fbLog.Error( sMessage := 'FB_SocketUdpCreate()', nErrID := fbCreate.nErrID );
				eStep := eUDP_STATE_ERROR;
			END_IF
		END_IF

	eUDP_STATE_SEND_START:
		fbSendTo( bExecute := FALSE );
		fbSendTo( sSrvNetId := sSrvNetId, sRemoteHost := stSendTo.stRemoteAddr.sAddr,
					nRemotePort := stSendTo.stRemoteAddr.nPort,
					pSrc:= ADR( stSendTo.txdata ),
					cbLen:= SIZEOF( stSendTo.txdata), 
					hSocket:= fbCreate.hSocket, bExecute:= TRUE );
					
     eStep := eUDP_STATE_SEND_WAIT;
	   	         
	eUDP_STATE_SEND_WAIT:
		fbSendTo( bExecute := FALSE );
		IF NOT fbSendTo.bBusy THEN
			IF NOT fbSendTo.bError THEN
				eStep := eUDP_STATE_RECEIVE_START;
			ELSE
				fbLog.Error( sMessage := 'FB_SocketUdpSendTo()', nErrID := fbSendTo.nErrID );
				eStep := eUDP_STATE_ERROR;
			END_IF
		END_IF

	eUDP_STATE_RECEIVE_START:
		MEMSET( ADR( stReceivedFrom ), 0, SIZEOF( stReceivedFrom ) );
		fbReceiveFrom( bExecute := FALSE );
		fbReceiveFrom( sSrvNetId := sSrvNetId, 
						pDest:= ADR( stReceivedFrom.rxdata ),
						cbLen:= SIZEOF( stReceivedFrom.rxdata ) - 1, (* Without string delimiter *)
						hSocket:= fbCreate.hSocket, bExecute:= TRUE );
		eStep := eUDP_STATE_RECEIVE_WAIT;

	eUDP_STATE_RECEIVE_WAIT:
		fbReceiveFrom( bExecute := FALSE );
		IF NOT fbReceiveFrom.bBusy THEN
			IF NOT fbReceiveFrom.bError THEN
				IF fbReceiveFrom.nRecBytes > 0 THEN
					
					stReceivedFrom.stRemoteAddr.sAddr := fbReceiveFrom.sRemoteHost;
					stReceivedFrom.stRemoteAddr.nPort := fbReceiveFrom.nRemotePort;
					
					fbRx.AddTail( stPut := stReceivedFrom );
					
					IF NOT fbRx.bOk THEN
						fbLog.Error( sMessage :='FB_FrameFifo(receiver)', nErrID := PLCPRJ_ERROR_RECFIFO_OVERFLOW );
					END_IF
				END_IF
				eStep := eUDP_STATE_IDLE;
			ELSE
				fbLog.Error( sMessage := 'FB_SocketUdpReceiveFrom()', nErrID := fbReceiveFrom.nErrID );
				IF fbReceiveFrom.nErrID = 16#80072746 THEN
					eStep := eUDP_STATE_IDLE;
				ELSE
					eStep := eUDP_STATE_ERROR;
				END_IF
			END_IF
		END_IF

	eUDP_STATE_CLOSE_START:
		fbLog.Message( sMessage := 'Closing connectionless (UDP) socket!', hSocket := fbCreate.hSocket );
		fbClose( bExecute := FALSE );
		fbClose( sSrvNetId := sSrvNetId, hSocket := fbCreate.hSocket, bExecute := TRUE );
		eStep := eUDP_STATE_CLOSE_WAIT;

	eUDP_STATE_CLOSE_WAIT:
		fbClose( bExecute := FALSE );
		IF NOT fbClose.bBusy THEN
			bCreated := FALSE;
			IF NOT fbClose.bError THEN
				eStep := eUDP_STATE_IDLE;
			ELSE
				fbLog.Error( sMessage := 'FB_SocketClose()', nErrID := fbClose.nErrID );
				eStep := eUDP_STATE_ERROR;
			END_IF
		END_IF

	eUDP_STATE_ERROR: 
		IF bCreated THEN
			eStep := eUDP_STATE_CLOSE_START;
		ELSE
			eStep := eUDP_STATE_IDLE;
		END_IF
END_CASE

END_FUNCTION_BLOCK

// ---- POUs/FUCTION BLOCK/UDP Source/FB_FrameFifo.TcPOU
FUNCTION_BLOCK FB_FrameFifo
VAR_INPUT
	bLog		: BOOL := FALSE;
	stPut		: ST_FrameFifoEntrydata;
	
END_VAR
VAR_OUTPUT
	bOk			: BOOL;
	stGet		: ST_FrameFifoEntrydata;
	nCount		: UDINT := 0;
END_VAR
VAR
	fbBuffer 	: FB_MemRingBuffer;
	buffer		: ARRAY[0..10000] OF BYTE;//ARRAY[0..NUMBER_OF_BYTE_FOR_ALL_FRAMEFIFO] OF BYTE;
	i : INT;
END_VAR
VAR CONSTANT
	SIZE_OF_FRAMEFIFO : UDINT := SIZEOF(ST_FrameFifoEntrydata);
	MAX_NUMBER_OF_FRAMEFIFO : UDINT := 10;
	NUMBER_OF_BYTE_FOR_ALL_FRAMEFIFO : UDINT := SIZE_OF_FRAMEFIFO*MAX_NUMBER_OF_FRAMEFIFO;
END_VAR

;

ACTION AddTail:

fbBuffer.A_AddTail( pBuffer:= ADR(buffer), cbBuffer:= SIZEOF(buffer),
					pWrite:= ADR( stPut ), cbWrite := SIZEOF( stPut ), 
					bOk=>bOk, nCount=>nCount );
END_ACTION

ACTION Clear:

FOR i:=0 TO TXDATASIZE BY 1 DO
stget.txdata[i] := 0; 
END_FOR

stGet.stRemoteAddr.nPort := 0;
stGet.stRemoteAddr.sAddr := '';
fbBuffer.A_Reset( pBuffer := ADR( buffer ), cbBuffer := SIZEOF( buffer ), 
					bOk=>bOk, nCount=>nCount );
END_ACTION

ACTION RemoveHead:

IF nCount = 0 THEN	 
FOR i:=0 TO TXDATASIZE BY 1 DO
stget.txdata[i] := 0;
END_FOR // clear


	stGet.stRemoteAddr.nPort := 0;
	stGet.stRemoteAddr.sAddr := '';
	bOk := FALSE;
	RETURN;
END_IF

fbBuffer.A_RemoveHead( pBuffer:= ADR(buffer), cbBuffer:= SIZEOF(buffer),
						pRead := ADR( stGet ), cbRead := SIZEOF( stGet ),
						bOk=>bOk, nCount=>nCount );
END_ACTION

END_FUNCTION_BLOCK

// ---- POUs/FUCTION BLOCK/UDP Source/FB_FrameFiforx.TcPOU
FUNCTION_BLOCK FB_FrameFiforx
VAR_INPUT
	bLog		: BOOL := FALSE;
	stPut		: ST_FrameFifoEntrydatarx;
	
END_VAR
VAR_OUTPUT
	bOk			: BOOL;
	stGet		: ST_FrameFifoEntrydatarx;
	nCount		: UDINT := 0;
END_VAR
VAR
	fbBuffer 	: FB_MemRingBuffer;
	buffer		: ARRAY[0..NUMBER_OF_BYTE_FOR_ALL_FRAMEFIFO] OF BYTE;
	i : INT;
END_VAR
VAR CONSTANT
	SIZE_OF_FRAMEFIFO : UDINT := SIZEOF(ST_FrameFifoEntrydatarx);
	MAX_NUMBER_OF_FRAMEFIFO : UDINT := 10;
	NUMBER_OF_BYTE_FOR_ALL_FRAMEFIFO : UDINT := SIZE_OF_FRAMEFIFO*MAX_NUMBER_OF_FRAMEFIFO;
END_VAR

ACTION AddTail:
fbBuffer.A_AddTail( pBuffer:= ADR(buffer), cbBuffer:= SIZEOF(buffer),
					pWrite:= ADR( stPut ), cbWrite := SIZEOF( stPut ), 
					bOk=>bOk, nCount=>nCount );
END_ACTION

ACTION Clear:
FOR i:=0 TO RXDATASIZE BY 1 DO
stGet.rxdata[i] := 0;
END_FOR 

stGet.stRemoteAddr.nPort := 0;
stGet.stRemoteAddr.sAddr := '';
fbBuffer.A_Reset( pBuffer := ADR( buffer ), cbBuffer := SIZEOF( buffer ), 
					bOk=>bOk, nCount=>nCount );
END_ACTION

ACTION RemoveHead:
IF nCount = 0 THEN
	 
FOR i:=0 TO RXDATASIZE BY 1 DO
stGet.rxdata[i] := 0;
END_FOR 

	stGet.stRemoteAddr.nPort := 0;
	stGet.stRemoteAddr.sAddr := '';
	bOk := FALSE;
	RETURN;
END_IF

fbBuffer.A_RemoveHead( pBuffer:= ADR(buffer), cbBuffer:= SIZEOF(buffer),
						pRead := ADR( stGet ), cbRead := SIZEOF( stGet ),
						bOk=>bOk, nCount=>nCount );
END_ACTION

END_FUNCTION_BLOCK

// ---- POUs/FUCTION BLOCK/UDP Source/FB_LogFifo.TcPOU
(* Log/debug/error message fifo *)
FUNCTION_BLOCK FB_LogFifo
VAR_INPUT
	bLog		: BOOL 		:= FALSE;(* TRUE => Enable log message output, FALSE => Disable *)
	sPrefix		: STRING 	:= 'Unknown::';(* Log message description string (allows the identification of log message source) *)
	
	sMessage	: STRING 	:= '';(* String message to add (write) to the fifo *)
	nErrID		: UDINT 	:= 0;(* Error code to add (write) to the fifo *)
	hSocket		: T_HSOCKET;(* Socket connection handle *)
END_VAR
VAR_OUTPUT
	bOk			: BOOL;(* TRUE = New entry added or removed succesfully, FALSE = Fifo overflow or fifo empty *)
	sGet		: T_MaxString := '';(* String entry removed (read) from fifo *)
	nCount		: UDINT := 0;(* Number of fifo entries *)
END_VAR
VAR
	fbBuffer 	: FB_StringRingBuffer;(* Basic (lower level) string buffer control function block *)
	buffer		: ARRAY[0..PLCPRJ_BUFFER_SIZE] OF BYTE;(* Internal buffer memory *)
	sSource		: T_MaxString;	
	sPut		: T_MaxString;
END_VAR

;

ACTION Clear:
(* Clears all fifo entries *)
fbBuffer.A_Reset( 	pBuffer := ADR( buffer ), cbBuffer := SIZEOF( buffer ), 
					bOk=>bOk, nCount=>nCount, getValue=>sGet );
END_ACTION

ACTION Error:
(* Adds new fifo entry *)
IF nErrID = 0 THEN
	sSource := '::Error: 0x';
ELSIF ( nErrID AND 16#80000000) = 16#80000000 THEN
	IF nErrID = 16#80072746 THEN
		sSource := '::Win32 error (the connection is reset by remote side): 0x';
	ELSE
		sSource := '::Win32 error: 0x';
	END_IF
ELSIF (nErrID AND 16#00008100) = 16#00008100 THEN
	CASE nErrID OF
		PLCPRJ_ERROR_SENDFIFO_OVERFLOW:
			sSource := '::PLC sample project send fifo overflow error: 0x';
		PLCPRJ_ERROR_RECFIFO_OVERFLOW:
			sSource := '::PLC sample project receive fifo overflow error: 0x';
	ELSE
		sSource := '::Other PLC sample project error: 0x';
	END_CASE
ELSIF (nErrID AND 16#00008000) = 16#00008000 THEN
	sSource := '::Internal TCP/IP Connection Server error: 0x';
ELSE
	sSource := '::TwinCAT System error: 0x';
END_IF

sPut := CONCAT( CONCAT( CONCAT( sPrefix, sMessage ), sSource ), DWORD_TO_HEXSTR( nErrID AND 16#FFFF, 0, FALSE ) ); 

fbBuffer.A_AddTail( pBuffer:= ADR(buffer), cbBuffer:= SIZEOF(buffer),
					putValue:= sPut, bOk=>bOk, nCount=>nCount );
IF bOk THEN
	IF bLog THEN(* Log error message *)
		ADSLOGSTR( ADSLOG_MSGTYPE_ERROR OR ADSLOG_MSGTYPE_LOG, '%s', sPut );	
	END_IF
END_IF
END_ACTION

ACTION Message:
(* Adds new fifo entry *)
sPut := CONCAT( CONCAT( sPrefix, sMessage ), CONCAT( '::', SOCKETADDR_TO_STRING(hSocket.localAddr) ) );
fbBuffer.A_AddTail( pBuffer:= ADR(buffer), cbBuffer:= SIZEOF(buffer),
					putValue:= sPut, bOk=>bOk, nCount=>nCount );
IF bOk THEN
	IF bLog THEN(* Log information message *)
		ADSLOGSTR( ADSLOG_MSGTYPE_HINT OR ADSLOG_MSGTYPE_LOG, '%s', sPut );	
	END_IF
END_IF
END_ACTION

ACTION Remove:
(* Removes oldest fifo entry *)
IF nCount = 0 THEN
	sGet := '';
	bOk := FALSE;
	RETURN;
END_IF

fbBuffer.A_RemoveHead( pBuffer:= ADR(buffer), cbBuffer:= SIZEOF(buffer),
						getValue=>sGet, bOk=>bOk, nCount=>nCount );
END_ACTION

END_FUNCTION_BLOCK

// ---- POUs/FUCTION BLOCK/UDP Source/FB_PeerToPeer_1.TcPOU

FUNCTION_BLOCK FB_PeerToPeer_1
VAR_IN_OUT
	
	fbTx	    : FB_FrameFifo_1;
	fbRx		: FB_FrameFiforx;
	fbLog		: FB_LogFifo;
	//bCreated		: BOOL;
END_VAR
VAR_INPUT
	sSrvNetId		: T_AmsNetID 	:= '';
	sLocalHost		: T_IPv4Addr 	:= '192.168.10.30';
	nLocalPort		: UDINT 		:= 53634;
	bEnable 		: BOOL			:= FALSE;
	tReconnect		: TIME			:= T#5S;
	bLog			: BOOL			:= FALSE;
	sPrefix			: STRING 		:= 'PeerToPeerX::';
	
	
END_VAR
VAR_OUTPUT
	bCreated		: BOOL;
END_VAR
VAR
	fbCreate		: FB_SocketUdpCreate;
	fbClose			: FB_SocketClose;
	fbReceiveFrom	: FB_SocketUdpReceiveFrom;
	fbSendTo		: FB_SocketUdpSendTo;
	
	stSendTo		: ST_FrameFifoEntrydata_1;
	stReceivedFrom	: ST_FrameFifoEntrydatarx;
	
	fbCreateTimer	: TON := ( PT := T#0S );	
	eStep			: E_ClientServerSteps;
	
	reseteventerror : BOOL; 
END_VAR

CASE eStep OF
	eUDP_STATE_IDLE:
		IF bEnable XOR bCreated THEN // XOR gate
			IF bEnable THEN
				fbTx.Clear( stput := stSendTo, bLog := bLog );
				fbRx.Clear( stput := stReceivedFrom, bLog := bLog );
				fbLog.Clear( sPrefix := sPrefix, bLog := bLog );

				fbCreateTimer( IN := TRUE );
				IF fbCreateTimer.Q THEN
					fbCreateTimer( IN := FALSE, PT := tReconnect ); 
					eStep := eUDP_STATE_CREATE_START;
				END_IF
			ELSE
				eStep := eUDP_STATE_CLOSE_START;
			END_IF
		ELSIF bCreated THEN
		fbTx.RemoveHead( stGet => stSendTo );
		IF fbTx.bok THEN
		   eStep := eUDP_STATE_SEND_START;
		ELSE 
		   eStep := eUDP_STATE_RECEIVE_START;  // Main receive peer to peer
		END_IF
	ELSE
		fbCreateTimer( IN := FALSE, PT := T#0S );
		END_IF

	eUDP_STATE_CREATE_START:
		fbCreate( bExecute := FALSE  );
		fbCreate( sSrvNetId := sSrvNetId, sLocalHost:= sLocalHost, nLocalPort:= nLocalPort, bExecute:= TRUE );
		eStep := eUDP_STATE_CREATE_WAIT;

	eUDP_STATE_CREATE_WAIT:
		fbCreate( bExecute := FALSE );
		IF NOT fbCreate.bBusy THEN
			IF NOT fbCreate.bError THEN
				bCreated := TRUE; // MAIN sequence
				fbLog.Message( sMessage := 'Connectionless (UDP) socket created!', hSocket := fbCreate.hSocket );
				eStep := eUDP_STATE_IDLE;
			ELSE
				fbLog.Error( sMessage := 'FB_SocketUdpCreate()', nErrID := fbCreate.nErrID );
				eStep := eUDP_STATE_ERROR;
			END_IF
		END_IF

	eUDP_STATE_SEND_START:
		fbSendTo( bExecute := FALSE );
		fbSendTo( sSrvNetId := sSrvNetId, sRemoteHost := stSendTo.stRemoteAddr.sAddr,
					nRemotePort := stSendTo.stRemoteAddr.nPort,
					pSrc:= ADR( stSendTo.txdata ),
					cbLen:= SIZEOF( stSendTo.txdata), 
					hSocket:= fbCreate.hSocket, bExecute:= TRUE );
					
     eStep := eUDP_STATE_SEND_WAIT;
	   	         
	eUDP_STATE_SEND_WAIT:
		fbSendTo( bExecute := FALSE );
		IF NOT fbSendTo.bBusy THEN
			IF NOT fbSendTo.bError THEN
				eStep := eUDP_STATE_RECEIVE_START;
			ELSE
				fbLog.Error( sMessage := 'FB_SocketUdpSendTo()', nErrID := fbSendTo.nErrID );
				eStep := eUDP_STATE_ERROR;
			END_IF
		END_IF

	eUDP_STATE_RECEIVE_START:
		MEMSET( ADR( stReceivedFrom ), 0, SIZEOF( stReceivedFrom ) );
		fbReceiveFrom( bExecute := FALSE );
		fbReceiveFrom( sSrvNetId := sSrvNetId, 
						pDest:= ADR( stReceivedFrom.rxdata ),
						cbLen:= SIZEOF( stReceivedFrom.rxdata ) - 1, (* Without string delimiter *)
						hSocket:= fbCreate.hSocket, bExecute:= TRUE );
		eStep := eUDP_STATE_RECEIVE_WAIT;

	eUDP_STATE_RECEIVE_WAIT:
		fbReceiveFrom( bExecute := FALSE );
		IF NOT fbReceiveFrom.bBusy THEN
			IF NOT fbReceiveFrom.bError THEN
				IF fbReceiveFrom.nRecBytes > 0 THEN
					
					stReceivedFrom.stRemoteAddr.sAddr := fbReceiveFrom.sRemoteHost;
					stReceivedFrom.stRemoteAddr.nPort := fbReceiveFrom.nRemotePort;
					
					fbRx.AddTail( stPut := stReceivedFrom );
					
					IF NOT fbRx.bOk THEN
						fbLog.Error( sMessage :='FB_FrameFifo(receiver)', nErrID := PLCPRJ_ERROR_RECFIFO_OVERFLOW );
					END_IF
				END_IF
				eStep := eUDP_STATE_IDLE;
			ELSE
				fbLog.Error( sMessage := 'FB_SocketUdpReceiveFrom()', nErrID := fbReceiveFrom.nErrID );
				IF fbReceiveFrom.nErrID = 16#80072746 THEN
					eStep := eUDP_STATE_IDLE;
				ELSE
					eStep := eUDP_STATE_ERROR;
				END_IF
			END_IF
		END_IF

	eUDP_STATE_CLOSE_START:
		fbLog.Message( sMessage := 'Closing connectionless (UDP) socket!', hSocket := fbCreate.hSocket );
		fbClose( bExecute := FALSE );
		fbClose( sSrvNetId := sSrvNetId, hSocket := fbCreate.hSocket, bExecute := TRUE );
		eStep := eUDP_STATE_CLOSE_WAIT;

	eUDP_STATE_CLOSE_WAIT:
		fbClose( bExecute := FALSE );
		IF NOT fbClose.bBusy THEN
			bCreated := FALSE;
			IF NOT fbClose.bError THEN
				eStep := eUDP_STATE_IDLE;
			ELSE
				fbLog.Error( sMessage := 'FB_SocketClose()', nErrID := fbClose.nErrID );
				eStep := eUDP_STATE_ERROR;
			END_IF
		END_IF

	eUDP_STATE_ERROR: 
		IF bCreated THEN
			eStep := eUDP_STATE_CLOSE_START;
		ELSE
			eStep := eUDP_STATE_IDLE;
		END_IF
END_CASE

END_FUNCTION_BLOCK

// ---- POUs/FUCTION BLOCK/UDP Source/FB_FrameFifo_1.TcPOU

FUNCTION_BLOCK FB_FrameFifo_1
VAR_INPUT
	bLog		: BOOL := FALSE;
	stPut		: ST_FrameFifoEntrydata_1;
	
END_VAR
VAR_OUTPUT
	bOk			: BOOL;
	stGet		: ST_FrameFifoEntrydata_1;
	nCount		: UDINT := 0;
END_VAR
VAR
	fbBuffer 	: FB_MemRingBuffer;
	buffer		: ARRAY[0..NUMBER_OF_BYTE_FOR_ALL_FRAMEFIFO] OF BYTE;
	i : INT;
END_VAR
VAR CONSTANT
	SIZE_OF_FRAMEFIFO : UDINT := SIZEOF(ST_FrameFifoEntrydata_1);
	MAX_NUMBER_OF_FRAMEFIFO : UDINT := 10;
	NUMBER_OF_BYTE_FOR_ALL_FRAMEFIFO : UDINT := SIZE_OF_FRAMEFIFO*MAX_NUMBER_OF_FRAMEFIFO;
END_VAR

;

ACTION AddTail:

fbBuffer.A_AddTail( pBuffer:= ADR(buffer), cbBuffer:= SIZEOF(buffer),
					pWrite:= ADR( stPut ), cbWrite := SIZEOF( stPut ), 
					bOk=>bOk, nCount=>nCount );
END_ACTION

ACTION Clear:

FOR i:=0 TO TXDATASIZE_1 BY 1 DO
stget.txdata[i] := 0; 
END_FOR

stGet.stRemoteAddr.nPort := 0;
stGet.stRemoteAddr.sAddr := '';
fbBuffer.A_Reset( pBuffer := ADR( buffer ), cbBuffer := SIZEOF( buffer ), 
					bOk=>bOk, nCount=>nCount );
END_ACTION

ACTION RemoveHead:
(* Removes oldest fifo entry *)
IF nCount = 0 THEN	 
FOR i:=0 TO TXDATASIZE_1 BY 1 DO
stget.txdata[i] := 0; 
END_FOR

	stGet.stRemoteAddr.nPort := 0;
	stGet.stRemoteAddr.sAddr := '';
	bOk := FALSE;
	RETURN;
END_IF

fbBuffer.A_RemoveHead( pBuffer:= ADR(buffer), cbBuffer:= SIZEOF(buffer),
						pRead := ADR( stGet ), cbRead := SIZEOF( stGet ),
						bOk=>bOk, nCount=>nCount );
END_ACTION

END_FUNCTION_BLOCK

// ---- POUs/FUCTION BLOCK/UDP Source/FB_PeerToPeer_2.TcPOU

FUNCTION_BLOCK FB_PeerToPeer_2
VAR_IN_OUT
	fbTx	    : FB_FrameFifo_2;
	fbRx		: FB_FrameFiforx;
	fbLog		: FB_LogFifo;
	//bCreated		: BOOL;
END_VAR
VAR_INPUT
	sSrvNetId		: T_AmsNetID 	:= '';
	sLocalHost		: T_IPv4Addr 	:= '192.168.10.30';
	nLocalPort		: UDINT 		:= 53634;
	bEnable 		: BOOL			:= FALSE;
	tReconnect		: TIME			:= T#5S;
	bLog			: BOOL			:= FALSE;
	sPrefix			: STRING 		:= 'PeerToPeerX::';
	
	
END_VAR
VAR_OUTPUT
	bCreated		: BOOL;
END_VAR
VAR
	fbCreate		: FB_SocketUdpCreate;
	fbClose			: FB_SocketClose;
	fbReceiveFrom	: FB_SocketUdpReceiveFrom;
	fbSendTo		: FB_SocketUdpSendTo;
	
	stSendTo		: ST_FrameFifoEntrydata_2;
	stReceivedFrom	: ST_FrameFifoEntrydatarx;
	
	fbCreateTimer	: TON := ( PT := T#0S );	
	eStep			: E_ClientServerSteps;
	
	reseteventerror : BOOL; 
END_VAR

CASE eStep OF
	eUDP_STATE_IDLE:
		IF bEnable XOR bCreated THEN
			IF bEnable THEN
				fbTx.Clear( stput := stSendTo, bLog := bLog );
				fbRx.Clear( stput := stReceivedFrom, bLog := bLog );
				fbLog.Clear( sPrefix := sPrefix, bLog := bLog );

				fbCreateTimer( IN := TRUE );
				IF fbCreateTimer.Q THEN
					fbCreateTimer( IN := FALSE, PT := tReconnect ); 
					eStep := eUDP_STATE_CREATE_START;
				END_IF
			ELSE
				eStep := eUDP_STATE_CLOSE_START;
			END_IF
		ELSIF bCreated THEN
		fbTx.RemoveHead( stGet => stSendTo );
		IF fbTx.bok THEN
		   eStep := eUDP_STATE_SEND_START;
		ELSE 
		   eStep := eUDP_STATE_RECEIVE_START; 
		END_IF 
	ELSE
		fbCreateTimer( IN := FALSE, PT := T#0S );
		END_IF

	eUDP_STATE_CREATE_START:
		fbCreate( bExecute := FALSE  );
		fbCreate( sSrvNetId := sSrvNetId, sLocalHost:= sLocalHost, nLocalPort:= nLocalPort, bExecute:= TRUE );
		eStep := eUDP_STATE_CREATE_WAIT;

	eUDP_STATE_CREATE_WAIT:
		fbCreate( bExecute := FALSE );
		IF NOT fbCreate.bBusy THEN
			IF NOT fbCreate.bError THEN
				bCreated := TRUE;
				fbLog.Message( sMessage := 'Connectionless (UDP) socket created!', hSocket := fbCreate.hSocket );
				eStep := eUDP_STATE_IDLE;
			ELSE
				fbLog.Error( sMessage := 'FB_SocketUdpCreate()', nErrID := fbCreate.nErrID );
				eStep := eUDP_STATE_ERROR;
			END_IF
		END_IF

	eUDP_STATE_SEND_START:
		fbSendTo( bExecute := FALSE );
		fbSendTo( sSrvNetId := sSrvNetId, sRemoteHost := stSendTo.stRemoteAddr.sAddr,
					nRemotePort := stSendTo.stRemoteAddr.nPort,
					pSrc:= ADR( stSendTo.txdata ),
					cbLen:= SIZEOF( stSendTo.txdata), 
					hSocket:= fbCreate.hSocket, bExecute:= TRUE );
					
     eStep := eUDP_STATE_SEND_WAIT;
	   	         
	eUDP_STATE_SEND_WAIT:
		fbSendTo( bExecute := FALSE );
		IF NOT fbSendTo.bBusy THEN
			IF NOT fbSendTo.bError THEN
				eStep := eUDP_STATE_RECEIVE_START;
			ELSE
				fbLog.Error( sMessage := 'FB_SocketUdpSendTo()', nErrID := fbSendTo.nErrID );
				eStep := eUDP_STATE_ERROR;
			END_IF
		END_IF

	eUDP_STATE_RECEIVE_START:
		MEMSET( ADR( stReceivedFrom ), 0, SIZEOF( stReceivedFrom ) );
		fbReceiveFrom( bExecute := FALSE );
		fbReceiveFrom( sSrvNetId := sSrvNetId, 
						pDest:= ADR( stReceivedFrom.rxdata ),
						cbLen:= SIZEOF( stReceivedFrom.rxdata ) - 1, (* Without string delimiter *)
						hSocket:= fbCreate.hSocket, bExecute:= TRUE );
		eStep := eUDP_STATE_RECEIVE_WAIT;

	eUDP_STATE_RECEIVE_WAIT:
		fbReceiveFrom( bExecute := FALSE );
		IF NOT fbReceiveFrom.bBusy THEN
			IF NOT fbReceiveFrom.bError THEN
				IF fbReceiveFrom.nRecBytes > 0 THEN
					
					stReceivedFrom.stRemoteAddr.sAddr := fbReceiveFrom.sRemoteHost;
					stReceivedFrom.stRemoteAddr.nPort := fbReceiveFrom.nRemotePort;
					
					fbRx.AddTail( stPut := stReceivedFrom );
					
					IF NOT fbRx.bOk THEN
						fbLog.Error( sMessage :='FB_FrameFifo(receiver)', nErrID := PLCPRJ_ERROR_RECFIFO_OVERFLOW );
					END_IF
				END_IF
				eStep := eUDP_STATE_IDLE;
			ELSE
				fbLog.Error( sMessage := 'FB_SocketUdpReceiveFrom()', nErrID := fbReceiveFrom.nErrID );
				IF fbReceiveFrom.nErrID = 16#80072746 THEN
					eStep := eUDP_STATE_IDLE;
				ELSE
					eStep := eUDP_STATE_ERROR;
				END_IF
			END_IF
		END_IF

	eUDP_STATE_CLOSE_START:
		fbLog.Message( sMessage := 'Closing connectionless (UDP) socket!', hSocket := fbCreate.hSocket );
		fbClose( bExecute := FALSE );
		fbClose( sSrvNetId := sSrvNetId, hSocket := fbCreate.hSocket, bExecute := TRUE );
		eStep := eUDP_STATE_CLOSE_WAIT;

	eUDP_STATE_CLOSE_WAIT:
		fbClose( bExecute := FALSE );
		IF NOT fbClose.bBusy THEN
			bCreated := FALSE;
			IF NOT fbClose.bError THEN
				eStep := eUDP_STATE_IDLE;
			ELSE
				fbLog.Error( sMessage := 'FB_SocketClose()', nErrID := fbClose.nErrID );
				eStep := eUDP_STATE_ERROR;
			END_IF
		END_IF

	eUDP_STATE_ERROR: 
		IF bCreated THEN
			eStep := eUDP_STATE_CLOSE_START;
		ELSE
			eStep := eUDP_STATE_IDLE;
		END_IF
END_CASE

END_FUNCTION_BLOCK

// ---- POUs/FUCTION BLOCK/UDP Source/FB_FrameFifo_2.TcPOU
FUNCTION_BLOCK FB_FrameFifo_2
VAR_INPUT
	bLog		: BOOL := FALSE;
	stPut		: ST_FrameFifoEntrydata_2;
	
END_VAR
VAR_OUTPUT
	bOk			: BOOL;
	stGet		: ST_FrameFifoEntrydata_2;
	nCount		: UDINT := 0;
END_VAR
VAR
	fbBuffer 	: FB_MemRingBuffer;
	buffer		: ARRAY[0..NUMBER_OF_BYTE_FOR_ALL_FRAMEFIFO] OF BYTE;
	i : INT;
END_VAR
VAR CONSTANT
	SIZE_OF_FRAMEFIFO : UDINT := SIZEOF(ST_FrameFifoEntrydata_2);
	MAX_NUMBER_OF_FRAMEFIFO : UDINT := 10;
	NUMBER_OF_BYTE_FOR_ALL_FRAMEFIFO : UDINT := SIZE_OF_FRAMEFIFO*MAX_NUMBER_OF_FRAMEFIFO;
END_VAR

;

ACTION AddTail:

fbBuffer.A_AddTail( pBuffer:= ADR(buffer), cbBuffer:= SIZEOF(buffer),
					pWrite:= ADR( stPut ), cbWrite := SIZEOF( stPut ), 
					bOk=>bOk, nCount=>nCount );
END_ACTION

ACTION Clear:

FOR i:=0 TO TXDATASIZE_2 BY 1 DO
stget.txdata[i] := 0;
END_FOR


stGet.stRemoteAddr.nPort := 0;
stGet.stRemoteAddr.sAddr := '';
fbBuffer.A_Reset( pBuffer := ADR( buffer ), cbBuffer := SIZEOF( buffer ), 
					bOk=>bOk, nCount=>nCount );
END_ACTION

ACTION RemoveHead:

IF nCount = 0 THEN	 

FOR i:=0 TO TXDATASIZE_2 BY 1 DO
stget.txdata[i] := 0;
END_FOR
	stGet.stRemoteAddr.nPort := 0;
	stGet.stRemoteAddr.sAddr := '';
	bOk := FALSE;
	RETURN;
END_IF

fbBuffer.A_RemoveHead( pBuffer:= ADR(buffer), cbBuffer:= SIZEOF(buffer),
						pRead := ADR( stGet ), cbRead := SIZEOF( stGet ),
						bOk=>bOk, nCount=>nCount );
END_ACTION

END_FUNCTION_BLOCK

// ---- POUs/FUNCTION/FC_HaversineDistance.TcPOU
FUNCTION FC_HaversineDistance : LREAL
VAR_INPUT
	lat1 : LREAL; // Current latitude
    lon1 : LREAL; // Current longitude
    lat2 : LREAL; // Target latitude
    lon2 : LREAL; // Target longitude
END_VAR
VAR
	 RR : LREAL := 6371000; // Radius of Earth in meters
    dLat, dLon, aa, cc : LREAL;
END_VAR

dLat := (lat2 - lat1) * PI / 180;
    dLon := (lon2 - lon1) * PI / 180;
    lat1 := lat1 * PI / 180;
    lat2 := lat2 * PI / 180;

    aa := SIN(dLat / 2) * SIN(dLat / 2) + COS(lat1) * COS(lat2) * SIN(dLon / 2) * SIN(dLon / 2);
    cc := 2 * ATAN(SQRT(aa) / SQRT(1 - aa));
    FC_HaversineDistance := (RR * cc);

END_FUNCTION

// ---- POUs/FUNCTION/FC_CalculateAzimuth.TcPOU
FUNCTION FC_CalculateAzimuth : LREAL
VAR_INPUT
	lat1 : LREAL; // Current latitude
    lon1 : LREAL; // Current longitude
    lat2 : LREAL; // Target latitude
    lon2 : LREAL; // Target longitude
END_VAR
VAR
	dLon, y, x, azimuth : LREAL;
END_VAR

 dLon := (lon2 - lon1) * PI / 180;
    lat1 := lat1 * PI / 180;
    lat2 := lat2 * PI / 180;

    y := SIN(dLon) * COS(lat2);
    x := COS(lat1) * SIN(lat2) - SIN(lat1) * COS(lat2) * COS(dLon);
    
    IF x = 0 THEN
        IF y > 0 THEN
            azimuth := 90;
        ELSIF y < 0 THEN
            azimuth := 270;
        ELSE
            azimuth := 0; // Undefined, but we set it to 0
        END_IF
    ELSE
        azimuth := ATAN(y / x) * 180 / PI;
        IF x < 0 THEN
            azimuth := azimuth + 180;
        ELSIF y < 0 THEN
            azimuth := azimuth + 360;
        END_IF
    END_IF
	
	IF azimuth >= 360 THEN
    azimuth := azimuth - 360;
    END_IF
    IF azimuth < 0 THEN
    azimuth := azimuth + 360;
     END_IF

    FC_CalculateAzimuth := azimuth;

END_FUNCTION
